LIN {X 0,Y 176.107,Z 395.866,A -85,B 0,C 180,E1 -22410,E2 -22410} C_VEL
LIN {X 0,Y 175.971,Z 396.64,A -85,B 0,C 180,E1 -22413.176,E2 -22413.176} C_VEL
LIN {X 0,Y 176.141,Z 396.55,A -85,B 0,C 180,E1 -22416.875,E2 -22416.875} C_VEL
LIN {X 0,Y 177.062,Z 394.985,A -85,B 0,C 180,E1 -22421.447,E2 -22421.447} C_VEL
LIN {X 0,Y 178.888,Z 391.863,A -85,B 0,C 180,E1 -22425.963,E2 -22425.963} C_VEL
LIN {X 0,Y 181.119,Z 388.376,A -85,B 0,C 180,E1 -22429.259,E2 -22429.259} C_VEL
LIN {X 0,Y 183.873,Z 383.839,A -85,B 0,C 180,E1 -22432.472,E2 -22432.472} C_VEL
LIN {X 0,Y 187.27,Z 377.805,A -85,B 0,C 180,E1 -22435.751,E2 -22435.751} C_VEL
LIN {X 0,Y 190.913,Z 371.032,A -85,B 0,C 180,E1 -22438.592,E2 -22438.592} C_VEL
LIN {X 0,Y 194.584,Z 363.85,A -85,B 0,C 180,E1 -22440.977,E2 -22440.977} C_VEL
LIN {X 0,Y 198.657,Z 355.185,A -85,B 0,C 180,E1 -22443.254,E2 -22443.254} C_VEL
LIN {X 0,Y 202.512,Z 345.804,A -85,B 0,C 180,E1 -22445.237,E2 -22445.237} C_VEL
LIN {X 0,Y 206.696,Z 334.241,A -85,B 0,C 180,E1 -22447.123,E2 -22447.123} C_VEL
LIN {X 0,Y 210.122,Z 322.779,A -85,B 0,C 180,E1 -22448.533,E2 -22448.533} C_VEL
LIN {X 0,Y 213.195,Z 309.844,A -85,B 0,C 180,E1 -22449.695,E2 -22449.695} C_VEL
LIN {X 0,Y 215.445,Z 296.998,A -85,B 0,C 180,E1 -22450.494,E2 -22450.494} C_VEL
LIN {X 0,Y 216.943,Z 281.701,A -85,B 0,C 180,E1 -22451.095,E2 -22451.095} C_VEL
LIN {X 0,Y 219.43,Z 248.273,A -85,B 0,C 180,E1 -22452.213,E2 -22452.213} C_VEL
LIN {X 0,Y 215.61,Z 238.212,A -85,B 0,C 180,E1 -22454.099,E2 -22454.099} C_VEL
LIN {X 0,Y 211.293,Z 228.849,A -85,B 0,C 180,E1 -22456.335,E2 -22456.335} C_VEL
LIN {X 0,Y 207.297,Z 221.367,A -85,B 0,C 180,E1 -22458.577,E2 -22458.577} C_VEL
LIN {X 0,Y 204.226,Z 216.042,A -85,B 0,C 180,E1 -22460.464,E2 -22460.464} C_VEL
LIN {X 0,Y 201.816,Z 212.042,A -85,B 0,C 180,E1 -22462.084,E2 -22462.084} C_VEL
LIN {X 0,Y 198.513,Z 206.797,A -85,B 0,C 180,E1 -22464.567,E2 -22464.567} C_VEL
LIN {X 0,Y 195.162,Z 201.691,A -85,B 0,C 180,E1 -22467.535,E2 -22467.535} C_VEL
LIN {X 0,Y 190.243,Z 194.896,A -85,B 0,C 180,E1 -22473.389,E2 -22473.389} C_VEL
LIN {X 0,Y 188.466,Z 192.868,A -85,B 0,C 180,E1 -22476.516,E2 -22476.516} C_VEL
LIN {X 0,Y 186.707,Z 191.554,A -85,B 0,C 180,E1 -22482.474,E2 -22482.474} C_VEL
LIN {X 0,Y 187.001,Z 191.732,A -85,B 0,C 180,E1 -22487.731,E2 -22487.731} C_VEL
LIN {X 0,Y 190.09,Z 193.411,A -85,B 0,C 180,E1 -22494.59,E2 -22494.59} C_VEL
LIN {X 0,Y 191.562,Z 196.122,A -85,B 0,C 180,E1 -22496.845,E2 -22496.845} C_VEL
LIN {X 0,Y 194.554,Z 198.965,A -85,B 0,C 180,E1 -22500.1,E2 -22500.1} C_VEL
LIN {X 0,Y 196.432,Z 202.226,A -85,B 0,C 180,E1 -22501.969,E2 -22501.969} C_VEL
LIN {X 0,Y 198.646,Z 204.552,A -85,B 0,C 180,E1 -22503.76,E2 -22503.76} C_VEL
LIN {X 0,Y 201.367,Z 208.221,A -85,B 0,C 180,E1 -22505.775,E2 -22505.775} C_VEL
LIN {X 0,Y 205.369,Z 214.172,A -85,B 0,C 180,E1 -22508.417,E2 -22508.417} C_VEL
LIN {X 0,Y 208.768,Z 219.318,A -85,B 0,C 180,E1 -22510.395,E2 -22510.395} C_VEL
LIN {X 0,Y 213.795,Z 228.478,A -85,B 0,C 180,E1 -22513.074,E2 -22513.074} C_VEL
LIN {X 0,Y 218.198,Z 237.802,A -85,B 0,C 180,E1 -22515.242,E2 -22515.242} C_VEL
LIN {X 0,Y 219.838,Z 242.158,A -85,B 0,C 180,E1 -22516.031,E2 -22516.031} C_VEL
LIN {X 0,Y 216.381,Z 285.399,A -85,B 0,C 180,E1 -22517.487,E2 -22517.487} C_VEL
LIN {X 0,Y 214.339,Z 299.301,A -85,B 0,C 180,E1 -22518.288,E2 -22518.288} C_VEL
LIN {X 0,Y 212.077,Z 310.584,A -85,B 0,C 180,E1 -22519.264,E2 -22519.264} C_VEL
LIN {X 0,Y 209.226,Z 321.582,A -85,B 0,C 180,E1 -22520.521,E2 -22520.521} C_VEL
LIN {X 0,Y 205.857,Z 332.053,A -85,B 0,C 180,E1 -22522.058,E2 -22522.058} C_VEL
LIN {X 0,Y 201.926,Z 342.352,A -85,B 0,C 180,E1 -22523.987,E2 -22523.987} C_VEL
LIN {X 0,Y 197.854,Z 351.744,A -85,B 0,C 180,E1 -22526.244,E2 -22526.244} C_VEL
LIN {X 0,Y 194.184,Z 359.384,A -85,B 0,C 180,E1 -22528.562,E2 -22528.562} C_VEL
LIN {X 0,Y 189.903,Z 367.38,A -85,B 0,C 180,E1 -22531.657,E2 -22531.657} C_VEL
LIN {X 0,Y 186.09,Z 373.869,A -85,B 0,C 180,E1 -22534.974,E2 -22534.974} C_VEL
LIN {X 0,Y 182.698,Z 379.213,A -85,B 0,C 180,E1 -22538.636,E2 -22538.636} C_VEL
LIN {X 0,Y 180.161,Z 382.905,A -85,B 0,C 180,E1 -22542.167,E2 -22542.167} C_VEL
LIN {X 0,Y 178.583,Z 385.029,A -85,B 0,C 180,E1 -22545.103,E2 -22545.103} C_VEL
LIN {X 0,Y 176.984,Z 386.777,A -85,B 0,C 180,E1 -22548.981,E2 -22548.981} C_VEL
LIN {X 0,Y 175.948,Z 387.352,A -85,B 0,C 180,E1 -22553.19,E2 -22553.19} C_VEL
LIN {X 0,Y 175.55,Z 386.619,A -85,B 0,C 180,E1 -22557.217,E2 -22557.217} C_VEL
LIN {X 0,Y 175.745,Z 384.409,A -85,B 0,C 180,E1 -22561.616,E2 -22561.616} C_VEL
LIN {X 0,Y 176.396,Z 381.454,A -85,B 0,C 180,E1 -22565.194,E2 -22565.194} C_VEL
LIN {X 0,Y 177.371,Z 376.912,A -85,B 0,C 180,E1 -22569.108,E2 -22569.108} C_VEL
LIN {X 0,Y 178.752,Z 371.021,A -85,B 0,C 180,E1 -22572.85,E2 -22572.85} C_VEL
LIN {X 0,Y 180.733,Z 363.522,A -85,B 0,C 180,E1 -22576.507,E2 -22576.507} C_VEL
LIN {X 0,Y 182.897,Z 355.757,A -85,B 0,C 180,E1 -22579.483,E2 -22579.483} C_VEL
LIN {X 0,Y 185.395,Z 346.038,A -85,B 0,C 180,E1 -22582.428,E2 -22582.428} C_VEL
LIN {X 0,Y 187.967,Z 335.639,A -85,B 0,C 180,E1 -22584.905,E2 -22584.905} C_VEL
LIN {X 0,Y 190.293,Z 324.879,A -85,B 0,C 180,E1 -22586.929,E2 -22586.929} C_VEL
LIN {X 0,Y 192.529,Z 312.621,A -85,B 0,C 180,E1 -22588.693,E2 -22588.693} C_VEL
LIN {X 0,Y 194.287,Z 300.473,A -85,B 0,C 180,E1 -22590,E2 -22590} C_VEL
LIN {X 0,Y 195.769,Z 287.395,A -85,B 0,C 180,E1 -22590.965,E2 -22590.965} C_VEL
LIN {X 0,Y 196.873,Z 270.105,A -85,B 0,C 180,E1 -22591.715,E2 -22591.715} C_VEL
LIN {X 0,Y 199.108,Z 225.699,A -85,B 0,C 180,E1 -22593.359,E2 -22593.359} C_VEL
LIN {X 0,Y 191.463,Z 205.022,A -85,B 0,C 180,E1 -22595.583,E2 -22595.583} C_VEL
LIN {X 0,Y 180.314,Z 184.581,A -85,B 0,C 180,E1 -22598.719,E2 -22598.719} C_VEL
LIN {X 0,Y 179.05,Z 182.009,A -85,B 0,C 180,E1 -22599.118,E2 -22599.118} C_VEL
LIN {X 0,Y 178.891,Z 181.212,A -85,B 0,C 180,E1 -22599.193,E2 -22599.193} C_VEL
LIN {X 0,Y 178.638,Z 181.233,A -85,B 0,C 180,E1 -22603.654,E2 -22603.654} C_VEL
LIN {X 0,Y 178.565,Z 181.241,A -85,B 0,C 180,E1 -22609.161,E2 -22609.161} C_VEL
LIN {X 0,Y 178.466,Z 181.238,A -85,B 0,C 180,E1 -22615.076,E2 -22615.076} C_VEL
LIN {X 0,Y 178.462,Z 181.246,A -85,B 0,C 180,E1 -22620.794,E2 -22620.794} C_VEL
LIN {X 0,Y 178.484,Z 181.225,A -85,B 0,C 180,E1 -22624.218,E2 -22624.218} C_VEL
LIN {X 0,Y 178.39,Z 181.264,A -85,B 0,C 180,E1 -22629.076,E2 -22629.076} C_VEL
LIN {X 0,Y 178.395,Z 181.255,A -85,B 0,C 180,E1 -22632.046,E2 -22632.046} C_VEL
LIN {X 0,Y 178.392,Z 181.224,A -85,B 0,C 180,E1 -22635.165,E2 -22635.165} C_VEL
LIN {X 0,Y 178.398,Z 181.233,A -85,B 0,C 180,E1 -22638.462,E2 -22638.462} C_VEL
LIN {X 0,Y 178.42,Z 181.26,A -85,B 0,C 180,E1 -22643.782,E2 -22643.782} C_VEL
LIN {X 0,Y 178.485,Z 181.245,A -85,B 0,C 180,E1 -22646.546,E2 -22646.546} C_VEL
LIN {X 0,Y 178.446,Z 181.256,A -85,B 0,C 180,E1 -22651.796,E2 -22651.796} C_VEL
LIN {X 0,Y 178.517,Z 181.241,A -85,B 0,C 180,E1 -22654.889,E2 -22654.889} C_VEL
LIN {X 0,Y 178.608,Z 181.235,A -85,B 0,C 180,E1 -22661.652,E2 -22661.652} C_VEL
LIN {X 0,Y 178.63,Z 181.221,A -85,B 0,C 180,E1 -22666.346,E2 -22666.346} C_VEL
LIN {X 0,Y 178.908,Z 181.197,A -85,B 0,C 180,E1 -22670.959,E2 -22670.959} C_VEL
LIN {X 0,Y 179.127,Z 181.171,A -85,B 0,C 180,E1 -22677.751,E2 -22677.751} C_VEL
LIN {X 0,Y 179.347,Z 181.143,A -85,B 0,C 180,E1 -22680,E2 -22680} C_VEL
LIN {X 0,Y 178.834,Z 181.175,A -85,B 0,C 180,E1 -22684.508,E2 -22684.508} C_VEL
LIN {X 0,Y 178.905,Z 181.171,A -85,B 0,C 180,E1 -22689.04,E2 -22689.04} C_VEL
LIN {X 0,Y 178.625,Z 181.235,A -85,B 0,C 180,E1 -22693.655,E2 -22693.655} C_VEL
LIN {X 0,Y 178.555,Z 181.214,A -85,B 0,C 180,E1 -22699.151,E2 -22699.151} C_VEL
LIN {X 0,Y 178.506,Z 181.248,A -85,B 0,C 180,E1 -22705.103,E2 -22705.103} C_VEL
LIN {X 0,Y 178.461,Z 181.256,A -85,B 0,C 180,E1 -22710.794,E2 -22710.794} C_VEL
LIN {X 0,Y 178.484,Z 181.249,A -85,B 0,C 180,E1 -22714.218,E2 -22714.218} C_VEL
LIN {X 0,Y 178.388,Z 181.265,A -85,B 0,C 180,E1 -22719.076,E2 -22719.076} C_VEL
LIN {X 0,Y 178.394,Z 181.262,A -85,B 0,C 180,E1 -22722.046,E2 -22722.046} C_VEL
LIN {X 0,Y 178.431,Z 181.452,A -85,B 0,C 180,E1 -22726.724,E2 -22726.724} C_VEL
LIN {X 0,Y 179.299,Z 184.858,A -85,B 0,C 180,E1 -22728.666,E2 -22728.666} C_VEL
LIN {X 0,Y 186.421,Z 200.095,A -85,B 0,C 180,E1 -22730.858,E2 -22730.858} C_VEL
LIN {X 0,Y 193.884,Z 218.787,A -85,B 0,C 180,E1 -22733.074,E2 -22733.074} C_VEL
LIN {X 0,Y 196.789,Z 227.908,A -85,B 0,C 180,E1 -22733.967,E2 -22733.967} C_VEL
LIN {X 0,Y 198.481,Z 242.952,A -85,B 0,C 180,E1 -22734.906,E2 -22734.906} C_VEL
LIN {X 0,Y 195.784,Z 293.869,A -85,B 0,C 180,E1 -22736.844,E2 -22736.844} C_VEL
LIN {X 0,Y 194.316,Z 307.658,A -85,B 0,C 180,E1 -22737.759,E2 -22737.759} C_VEL
LIN {X 0,Y 193.602,Z 312.687,A -85,B 0,C 180,E1 -22738.205,E2 -22738.205} C_VEL
LIN {X 0,Y 192.145,Z 318.194,A -85,B 0,C 180,E1 -22738.68,E2 -22738.68} C_VEL
LIN {X 0,Y 188.016,Z 326.878,A -85,B 0,C 180,E1 -22739.416,E2 -22739.416} C_VEL
LIN {X 0,Y 183.577,Z 335.199,A -85,B 0,C 180,E1 -22740.384,E2 -22740.384} C_VEL
LIN {X 0,Y 181.663,Z 340.142,A -85,B 0,C 180,E1 -22741.217,E2 -22741.217} C_VEL
LIN {X 0,Y 179.121,Z 350.496,A -85,B 0,C 180,E1 -22743.493,E2 -22743.493} C_VEL
LIN {X 0,Y 176.758,Z 359.609,A -85,B 0,C 180,E1 -22746.012,E2 -22746.012} C_VEL
LIN {X 0,Y 175.261,Z 365.095,A -85,B 0,C 180,E1 -22747.815,E2 -22747.815} C_VEL
LIN {X 0,Y 173.041,Z 373.154,A -85,B 0,C 180,E1 -22751.039,E2 -22751.039} C_VEL
LIN {X 0,Y 171.159,Z 380.029,A -85,B 0,C 180,E1 -22754.52,E2 -22754.52} C_VEL
LIN {X 0,Y 169.97,Z 385.517,A -85,B 0,C 180,E1 -22758.068,E2 -22758.068} C_VEL
LIN {X 0,Y 169.249,Z 389.772,A -85,B 0,C 180,E1 -22761.643,E2 -22761.643} C_VEL
LIN {X 0,Y 168.931,Z 392.919,A -85,B 0,C 180,E1 -22765.227,E2 -22765.227} C_VEL
LIN {X 0,Y 168.947,Z 394.472,A -85,B 0,C 180,E1 -22767.616,E2 -22767.616} C_VEL
LIN {X 0,Y 169.015,Z 395.567,A -85,B 0,C 180,E1 -22770,E2 -22770} C_VEL
LIN {X 0,Y 168.892,Z 396.323,A -85,B 0,C 180,E1 -22772.921,E2 -22772.921} C_VEL
LIN {X 0,Y 169.093,Z 396.381,A -85,B 0,C 180,E1 -22777.163,E2 -22777.163} C_VEL
LIN {X 0,Y 169.462,Z 395.868,A -85,B 0,C 180,E1 -22779.549,E2 -22779.549} C_VEL
LIN {X 0,Y 170.961,Z 393.626,A -85,B 0,C 180,E1 -22784.28,E2 -22784.28} C_VEL
LIN {X 0,Y 172.77,Z 390.889,A -85,B 0,C 180,E1 -22787.764,E2 -22787.764} C_VEL
LIN {X 0,Y 175.373,Z 387.162,A -85,B 0,C 180,E1 -22791.142,E2 -22791.142} C_VEL
LIN {X 0,Y 178.401,Z 382.356,A -85,B 0,C 180,E1 -22794.434,E2 -22794.434} C_VEL
LIN {X 0,Y 182.612,Z 375.225,A -85,B 0,C 180,E1 -22798.129,E2 -22798.129} C_VEL
LIN {X 0,Y 186.944,Z 367.53,A -85,B 0,C 180,E1 -22801.126,E2 -22801.126} C_VEL
LIN {X 0,Y 191.916,Z 357.942,A -85,B 0,C 180,E1 -22803.95,E2 -22803.95} C_VEL
LIN {X 0,Y 196.347,Z 348.123,A -85,B 0,C 180,E1 -22806.2,E2 -22806.2} C_VEL
LIN {X 0,Y 200.691,Z 337.124,A -85,B 0,C 180,E1 -22808.113,E2 -22808.113} C_VEL
LIN {X 0,Y 204.719,Z 324.761,A -85,B 0,C 180,E1 -22809.747,E2 -22809.747} C_VEL
LIN {X 0,Y 207.863,Z 312.663,A -85,B 0,C 180,E1 -22810.926,E2 -22810.926} C_VEL
LIN {X 0,Y 210.488,Z 299.25,A -85,B 0,C 180,E1 -22811.816,E2 -22811.816} C_VEL
LIN {X 0,Y 212.045,Z 286.37,A -85,B 0,C 180,E1 -22812.391,E2 -22812.391} C_VEL
LIN {X 0,Y 214.842,Z 250.537,A -85,B 0,C 180,E1 -22813.61,E2 -22813.61} C_VEL
LIN {X 0,Y 211.062,Z 240.778,A -85,B 0,C 180,E1 -22815.632,E2 -22815.632} C_VEL
LIN {X 0,Y 206.868,Z 231.538,A -85,B 0,C 180,E1 -22818.017,E2 -22818.017} C_VEL
LIN {X 0,Y 202.25,Z 222.91,A -85,B 0,C 180,E1 -22820.911,E2 -22820.911} C_VEL
LIN {X 0,Y 199.146,Z 217.613,A -85,B 0,C 180,E1 -22823.134,E2 -22823.134} C_VEL
LIN {X 0,Y 196.249,Z 212.847,A -85,B 0,C 180,E1 -22825.454,E2 -22825.454} C_VEL
LIN {X 0,Y 192.831,Z 207.539,A -85,B 0,C 180,E1 -22828.749,E2 -22828.749} C_VEL
LIN {X 0,Y 188.741,Z 201.564,A -85,B 0,C 180,E1 -22834.1,E2 -22834.1} C_VEL
LIN {X 0,Y 187.288,Z 199.823,A -85,B 0,C 180,E1 -22836.895,E2 -22836.895} C_VEL
LIN {X 0,Y 185.731,Z 198.59,A -85,B 0,C 180,E1 -22842.379,E2 -22842.379} C_VEL
LIN {X 0,Y 186.009,Z 198.77,A -85,B 0,C 180,E1 -22847.752,E2 -22847.752} C_VEL
LIN {X 0,Y 188.742,Z 200.32,A -85,B 0,C 180,E1 -22854.119,E2 -22854.119} C_VEL
LIN {X 0,Y 190.143,Z 202.883,A -85,B 0,C 180,E1 -22856.351,E2 -22856.351} C_VEL
LIN {X 0,Y 192.838,Z 205.635,A -85,B 0,C 180,E1 -22859.478,E2 -22859.478} C_VEL
LIN {X 0,Y 194.729,Z 208.869,A -85,B 0,C 180,E1 -22861.431,E2 -22861.431} C_VEL
LIN {X 0,Y 196.672,Z 211.096,A -85,B 0,C 180,E1 -22863.118,E2 -22863.118} C_VEL
LIN {X 0,Y 199.963,Z 215.717,A -85,B 0,C 180,E1 -22865.637,E2 -22865.637} C_VEL
LIN {X 0,Y 204.862,Z 223.149,A -85,B 0,C 180,E1 -22868.874,E2 -22868.874} C_VEL
LIN {X 0,Y 208.76,Z 230.33,A -85,B 0,C 180,E1 -22871.187,E2 -22871.187} C_VEL
LIN {X 0,Y 212.936,Z 238.93,A -85,B 0,C 180,E1 -22873.425,E2 -22873.425} C_VEL
LIN {X 0,Y 215.288,Z 244.559,A -85,B 0,C 180,E1 -22874.639,E2 -22874.639} C_VEL
LIN {X 0,Y 211.784,Z 285.821,A -85,B 0,C 180,E1 -22876.042,E2 -22876.042} C_VEL
LIN {X 0,Y 209.706,Z 299.278,A -85,B 0,C 180,E1 -22876.818,E2 -22876.818} C_VEL
LIN {X 0,Y 207.25,Z 311.125,A -85,B 0,C 180,E1 -22877.853,E2 -22877.853} C_VEL
LIN {X 0,Y 203.846,Z 323.371,A -85,B 0,C 180,E1 -22879.297,E2 -22879.297} C_VEL
LIN {X 0,Y 199.706,Z 335.316,A -85,B 0,C 180,E1 -22881.158,E2 -22881.158} C_VEL
LIN {X 0,Y 195.305,Z 345.853,A -85,B 0,C 180,E1 -22883.318,E2 -22883.318} C_VEL
LIN {X 0,Y 191.287,Z 354.267,A -85,B 0,C 180,E1 -22885.521,E2 -22885.521} C_VEL
LIN {X 0,Y 187.201,Z 361.997,A -85,B 0,C 180,E1 -22888.084,E2 -22888.084} C_VEL
LIN {X 0,Y 182.843,Z 369.539,A -85,B 0,C 180,E1 -22891.316,E2 -22891.316} C_VEL
LIN {X 0,Y 179.147,Z 375.283,A -85,B 0,C 180,E1 -22894.528,E2 -22894.528} C_VEL
LIN {X 0,Y 175.416,Z 380.612,A -85,B 0,C 180,E1 -22898.623,E2 -22898.623} C_VEL
LIN {X 0,Y 172.573,Z 384.364,A -85,B 0,C 180,E1 -22902.857,E2 -22902.857} C_VEL
LIN {X 0,Y 171.125,Z 386.009,A -85,B 0,C 180,E1 -22905.718,E2 -22905.718} C_VEL
LIN {X 0,Y 170.001,Z 387.077,A -85,B 0,C 180,E1 -22908.589,E2 -22908.589} C_VEL
LIN {X 0,Y 169.019,Z 387.547,A -85,B 0,C 180,E1 -22912.19,E2 -22912.19} C_VEL
LIN {X 0,Y 168.488,Z 386.939,A -85,B 0,C 180,E1 -22916.537,E2 -22916.537} C_VEL
LIN {X 0,Y 168.576,Z 384.833,A -85,B 0,C 180,E1 -22921.105,E2 -22921.105} C_VEL
LIN {X 0,Y 169.348,Z 381.387,A -85,B 0,C 180,E1 -22925.48,E2 -22925.48} C_VEL
LIN {X 0,Y 170.352,Z 376.838,A -85,B 0,C 180,E1 -22929.471,E2 -22929.471} C_VEL
LIN {X 0,Y 171.814,Z 370.863,A -85,B 0,C 180,E1 -22933.361,E2 -22933.361} C_VEL
LIN {X 0,Y 173.965,Z 363.113,A -85,B 0,C 180,E1 -22937.235,E2 -22937.235} C_VEL
LIN {X 0,Y 176.178,Z 355.408,A -85,B 0,C 180,E1 -22940.239,E2 -22940.239} C_VEL
LIN {X 0,Y 178.778,Z 345.747,A -85,B 0,C 180,E1 -22943.227,E2 -22943.227} C_VEL
LIN {X 0,Y 181.436,Z 335.304,A -85,B 0,C 180,E1 -22945.772,E2 -22945.772} C_VEL
LIN {X 0,Y 183.793,Z 324.677,A -85,B 0,C 180,E1 -22947.808,E2 -22947.808} C_VEL
LIN {X 0,Y 186.077,Z 312.539,A -85,B 0,C 180,E1 -22949.594,E2 -22949.594} C_VEL
LIN {X 0,Y 187.926,Z 300.289,A -85,B 0,C 180,E1 -22950.937,E2 -22950.937} C_VEL
LIN {X 0,Y 189.456,Z 286.987,A -85,B 0,C 180,E1 -22951.927,E2 -22951.927} C_VEL
LIN {X 0,Y 190.6,Z 269.299,A -85,B 0,C 180,E1 -22952.701,E2 -22952.701} C_VEL
LIN {X 0,Y 192.875,Z 227.779,A -85,B 0,C 180,E1 -22954.266,E2 -22954.266} C_VEL
LIN {X 0,Y 185.991,Z 208.623,A -85,B 0,C 180,E1 -22956.403,E2 -22956.403} C_VEL
LIN {X 0,Y 174.96,Z 188.375,A -85,B 0,C 180,E1 -22959.659,E2 -22959.659} C_VEL
LIN {X 0,Y 173.38,Z 185.708,A -85,B 0,C 180,E1 -22960.157,E2 -22960.157} C_VEL
LIN {X 0,Y 172.041,Z 183.219,A -85,B 0,C 180,E1 -22960.601,E2 -22960.601} C_VEL
LIN {X 0,Y 171.798,Z 182.075,A -85,B 0,C 180,E1 -22960.758,E2 -22960.758} C_VEL
LIN {X 0,Y 171.517,Z 182.104,A -85,B 0,C 180,E1 -22966.668,E2 -22966.668} C_VEL
LIN {X 0,Y 171.491,Z 182.124,A -85,B 0,C 180,E1 -22969.51,E2 -22969.51} C_VEL
LIN {X 0,Y 171.404,Z 182.121,A -85,B 0,C 180,E1 -22975.57,E2 -22975.57} C_VEL
LIN {X 0,Y 171.419,Z 182.125,A -85,B 0,C 180,E1 -22980.573,E2 -22980.573} C_VEL
LIN {X 0,Y 171.393,Z 182.112,A -85,B 0,C 180,E1 -22985.035,E2 -22985.035} C_VEL
LIN {X 0,Y 171.353,Z 182.14,A -85,B 0,C 180,E1 -22988.805,E2 -22988.805} C_VEL
LIN {X 0,Y 171.319,Z 182.113,A -85,B 0,C 180,E1 -22994.218,E2 -22994.218} C_VEL
LIN {X 0,Y 171.331,Z 182.118,A -85,B 0,C 180,E1 -22998.98,E2 -22998.98} C_VEL
LIN {X 0,Y 171.361,Z 182.136,A -85,B 0,C 180,E1 -23002.034,E2 -23002.034} C_VEL
LIN {X 0,Y 171.399,Z 182.133,A -85,B 0,C 180,E1 -23005.093,E2 -23005.093} C_VEL
LIN {X 0,Y 171.411,Z 182.129,A -85,B 0,C 180,E1 -23010.527,E2 -23010.527} C_VEL
LIN {X 0,Y 171.438,Z 182.119,A -85,B 0,C 180,E1 -23015.798,E2 -23015.798} C_VEL
LIN {X 0,Y 171.509,Z 182.121,A -85,B 0,C 180,E1 -23020.863,E2 -23020.863} C_VEL
LIN {X 0,Y 171.545,Z 182.101,A -85,B 0,C 180,E1 -23025.77,E2 -23025.77} C_VEL
LIN {X 0,Y 171.846,Z 182.078,A -85,B 0,C 180,E1 -23030.585,E2 -23030.585} C_VEL
LIN {X 0,Y 171.787,Z 182.077,A -85,B 0,C 180,E1 -23035.307,E2 -23035.307} C_VEL
LIN {X 0,Y 172.312,Z 182.019,A -85,B 0,C 180,E1 -23040,E2 -23040} C_VEL
LIN {X 0,Y 171.783,Z 182.048,A -85,B 0,C 180,E1 -23044.693,E2 -23044.693} C_VEL
LIN {X 0,Y 171.844,Z 182.054,A -85,B 0,C 180,E1 -23049.415,E2 -23049.415} C_VEL
LIN {X 0,Y 171.541,Z 182.117,A -85,B 0,C 180,E1 -23054.23,E2 -23054.23} C_VEL
LIN {X 0,Y 171.479,Z 182.092,A -85,B 0,C 180,E1 -23059.498,E2 -23059.498} C_VEL
LIN {X 0,Y 171.436,Z 182.131,A -85,B 0,C 180,E1 -23065.592,E2 -23065.592} C_VEL
LIN {X 0,Y 171.419,Z 182.133,A -85,B 0,C 180,E1 -23070.572,E2 -23070.572} C_VEL
LIN {X 0,Y 171.393,Z 182.135,A -85,B 0,C 180,E1 -23075.035,E2 -23075.035} C_VEL
LIN {X 0,Y 171.344,Z 182.143,A -85,B 0,C 180,E1 -23078.801,E2 -23078.801} C_VEL
LIN {X 0,Y 171.319,Z 182.137,A -85,B 0,C 180,E1 -23084.218,E2 -23084.218} C_VEL
LIN {X 0,Y 171.386,Z 182.139,A -85,B 0,C 180,E1 -23085.599,E2 -23085.599} C_VEL
LIN {X 0,Y 171.959,Z 184.583,A -85,B 0,C 180,E1 -23087.052,E2 -23087.052} C_VEL
LIN {X 0,Y 178.775,Z 198.802,A -85,B 0,C 180,E1 -23089.287,E2 -23089.287} C_VEL
LIN {X 0,Y 185.122,Z 213.873,A -85,B 0,C 180,E1 -23091.293,E2 -23091.293} C_VEL
LIN {X 0,Y 190.538,Z 228.94,A -85,B 0,C 180,E1 -23092.988,E2 -23092.988} C_VEL
LIN {X 0,Y 192.183,Z 243.751,A -85,B 0,C 180,E1 -23093.956,E2 -23093.956} C_VEL
LIN {X 0,Y 189.431,Z 293.655,A -85,B 0,C 180,E1 -23095.91,E2 -23095.91} C_VEL
LIN {X 0,Y 187.93,Z 307.365,A -85,B 0,C 180,E1 -23096.843,E2 -23096.843} C_VEL
LIN {X 0,Y 186.046,Z 319.586,A -85,B 0,C 180,E1 -23098.071,E2 -23098.071} C_VEL
LIN {X 0,Y 183.534,Z 332.205,A -85,B 0,C 180,E1 -23099.828,E2 -23099.828} C_VEL
LIN {X 0,Y 181.663,Z 340.142,A -85,B 0,C 180,E1 -23101.217,E2 -23101.217} C_VEL
LIN {X 0,Y 179.676,Z 345.025,A -85,B 0,C 180,E1 -23102.13,E2 -23102.13} C_VEL
LIN {X 0,Y 172.868,Z 355.309,A -85,B 0,C 180,E1 -23104.252,E2 -23104.252} C_VEL
LIN {X 0,Y 169.601,Z 360.842,A -85,B 0,C 180,E1 -23105.784,E2 -23105.784} C_VEL
LIN {X 0,Y 168.69,Z 363.503,A -85,B 0,C 180,E1 -23106.693,E2 -23106.693} C_VEL
LIN {X 0,Y 167.072,Z 369.581,A -85,B 0,C 180,E1 -23109.05,E2 -23109.05} C_VEL
LIN {X 0,Y 164.926,Z 377.141,A -85,B 0,C 180,E1 -23112.645,E2 -23112.645} C_VEL
LIN {X 0,Y 163.342,Z 383.188,A -85,B 0,C 180,E1 -23116.311,E2 -23116.311} C_VEL
LIN {X 0,Y 162.414,Z 387.947,A -85,B 0,C 180,E1 -23120.033,E2 -23120.033} C_VEL
LIN {X 0,Y 161.906,Z 391.539,A -85,B 0,C 180,E1 -23123.77,E2 -23123.77} C_VEL
LIN {X 0,Y 161.866,Z 394.085,A -85,B 0,C 180,E1 -23127.512,E2 -23127.512} C_VEL
LIN {X 0,Y 161.924,Z 395.256,A -85,B 0,C 180,E1 -23130,E2 -23130} C_VEL
LIN {X 0,Y 161.797,Z 395.963,A -85,B 0,C 180,E1 -23132.49,E2 -23132.49} C_VEL
LIN {X 0,Y 161.85,Z 396.276,A -85,B 0,C 180,E1 -23134.982,E2 -23134.982} C_VEL
LIN {X 0,Y 162.44,Z 395.758,A -85,B 0,C 180,E1 -23139.966,E2 -23139.966} C_VEL
LIN {X 0,Y 163.131,Z 394.899,A -85,B 0,C 180,E1 -23142.44,E2 -23142.44} C_VEL
LIN {X 0,Y 165.232,Z 391.971,A -85,B 0,C 180,E1 -23147.322,E2 -23147.322} C_VEL
LIN {X 0,Y 167.763,Z 388.674,A -85,B 0,C 180,E1 -23150.86,E2 -23150.86} C_VEL
LIN {X 0,Y 170.809,Z 384.361,A -85,B 0,C 180,E1 -23154.296,E2 -23154.296} C_VEL
LIN {X 0,Y 174.933,Z 378.091,A -85,B 0,C 180,E1 -23158.048,E2 -23158.048} C_VEL
LIN {X 0,Y 179.394,Z 370.883,A -85,B 0,C 180,E1 -23161.271,E2 -23161.271} C_VEL
LIN {X 0,Y 183.502,Z 363.774,A -85,B 0,C 180,E1 -23163.735,E2 -23163.735} C_VEL
LIN {X 0,Y 187.957,Z 355.211,A -85,B 0,C 180,E1 -23166.08,E2 -23166.08} C_VEL
LIN {X 0,Y 192.215,Z 345.901,A -85,B 0,C 180,E1 -23168.098,E2 -23168.098} C_VEL
LIN {X 0,Y 196.761,Z 334.474,A -85,B 0,C 180,E1 -23170.011,E2 -23170.011} C_VEL
LIN {X 0,Y 200.465,Z 323.297,A -85,B 0,C 180,E1 -23171.432,E2 -23171.432} C_VEL
LIN {X 0,Y 203.774,Z 310.711,A -85,B 0,C 180,E1 -23172.598,E2 -23172.598} C_VEL
LIN {X 0,Y 206.365,Z 297.392,A -85,B 0,C 180,E1 -23173.453,E2 -23173.453} C_VEL
LIN {X 0,Y 207.997,Z 282.871,A -85,B 0,C 180,E1 -23174.052,E2 -23174.052} C_VEL
LIN {X 0,Y 210.445,Z 253.266,A -85,B 0,C 180,E1 -23175.05,E2 -23175.05} C_VEL
LIN {X 0,Y 207.149,Z 244.462,A -85,B 0,C 180,E1 -23176.956,E2 -23176.956} C_VEL
LIN {X 0,Y 203.33,Z 235.89,A -85,B 0,C 180,E1 -23179.332,E2 -23179.332} C_VEL
LIN {X 0,Y 199.096,Z 227.688,A -85,B 0,C 180,E1 -23182.237,E2 -23182.237} C_VEL
LIN {X 0,Y 196.6,Z 223.285,A -85,B 0,C 180,E1 -23184.167,E2 -23184.167} C_VEL
LIN {X 0,Y 194.365,Z 219.331,A -85,B 0,C 180,E1 -23186.106,E2 -23186.106} C_VEL
LIN {X 0,Y 191.155,Z 214.149,A -85,B 0,C 180,E1 -23189.363,E2 -23189.363} C_VEL
LIN {X 0,Y 187.361,Z 208.322,A -85,B 0,C 180,E1 -23194.669,E2 -23194.669} C_VEL
LIN {X 0,Y 186.118,Z 206.776,A -85,B 0,C 180,E1 -23197.279,E2 -23197.279} C_VEL
LIN {X 0,Y 184.756,Z 205.624,A -85,B 0,C 180,E1 -23202.283,E2 -23202.283} C_VEL
LIN {X 0,Y 185.007,Z 205.776,A -85,B 0,C 180,E1 -23207.685,E2 -23207.685} C_VEL
LIN {X 0,Y 187.517,Z 207.361,A -85,B 0,C 180,E1 -23213.812,E2 -23213.812} C_VEL
LIN {X 0,Y 189.221,Z 210.259,A -85,B 0,C 180,E1 -23216.523,E2 -23216.523} C_VEL
LIN {X 0,Y 191.172,Z 212.351,A -85,B 0,C 180,E1 -23218.881,E2 -23218.881} C_VEL
LIN {X 0,Y 193.376,Z 215.915,A -85,B 0,C 180,E1 -23221.2,E2 -23221.2} C_VEL
LIN {X 0,Y 194.887,Z 217.786,A -85,B 0,C 180,E1 -23222.565,E2 -23222.565} C_VEL
LIN {X 0,Y 197.754,Z 221.997,A -85,B 0,C 180,E1 -23224.895,E2 -23224.895} C_VEL
LIN {X 0,Y 202.144,Z 228.943,A -85,B 0,C 180,E1 -23227.994,E2 -23227.994} C_VEL
LIN {X 0,Y 205.659,Z 235.617,A -85,B 0,C 180,E1 -23230.199,E2 -23230.199} C_VEL
LIN {X 0,Y 209.687,Z 244.391,A -85,B 0,C 180,E1 -23232.533,E2 -23232.533} C_VEL
LIN {X 0,Y 210.887,Z 247.219,A -85,B 0,C 180,E1 -23233.186,E2 -23233.186} C_VEL
LIN {X 0,Y 207.416,Z 286.223,A -85,B 0,C 180,E1 -23234.52,E2 -23234.52} C_VEL
LIN {X 0,Y 205.186,Z 299.973,A -85,B 0,C 180,E1 -23235.319,E2 -23235.319} C_VEL
LIN {X 0,Y 202.714,Z 311.154,A -85,B 0,C 180,E1 -23236.299,E2 -23236.299} C_VEL
LIN {X 0,Y 199.234,Z 323.283,A -85,B 0,C 180,E1 -23237.742,E2 -23237.742} C_VEL
LIN {X 0,Y 195.19,Z 334.464,A -85,B 0,C 180,E1 -23239.471,E2 -23239.471} C_VEL
LIN {X 0,Y 190.532,Z 345.267,A -85,B 0,C 180,E1 -23241.646,E2 -23241.646} C_VEL
LIN {X 0,Y 186.342,Z 353.743,A -85,B 0,C 180,E1 -23243.849,E2 -23243.849} C_VEL
LIN {X 0,Y 181.27,Z 362.828,A -85,B 0,C 180,E1 -23246.907,E2 -23246.907} C_VEL
LIN {X 0,Y 176.91,Z 369.861,A -85,B 0,C 180,E1 -23250.013,E2 -23250.013} C_VEL
LIN {X 0,Y 172.79,Z 375.846,A -85,B 0,C 180,E1 -23253.507,E2 -23253.507} C_VEL
LIN {X 0,Y 168.831,Z 381.067,A -85,B 0,C 180,E1 -23257.727,E2 -23257.727} C_VEL
LIN {X 0,Y 166.726,Z 383.673,A -85,B 0,C 180,E1 -23260.645,E2 -23260.645} C_VEL
LIN {X 0,Y 164.978,Z 385.602,A -85,B 0,C 180,E1 -23263.598,E2 -23263.598} C_VEL
LIN {X 0,Y 163.414,Z 387.024,A -85,B 0,C 180,E1 -23266.981,E2 -23266.981} C_VEL
LIN {X 0,Y 162.113,Z 387.737,A -85,B 0,C 180,E1 -23271.293,E2 -23271.293} C_VEL
LIN {X 0,Y 161.422,Z 387.22,A -85,B 0,C 180,E1 -23275.815,E2 -23275.815} C_VEL
LIN {X 0,Y 161.423,Z 385.243,A -85,B 0,C 180,E1 -23280.547,E2 -23280.547} C_VEL
LIN {X 0,Y 162.004,Z 382.624,A -85,B 0,C 180,E1 -23284.29,E2 -23284.29} C_VEL
LIN {X 0,Y 162.951,Z 378.413,A -85,B 0,C 180,E1 -23288.494,E2 -23288.494} C_VEL
LIN {X 0,Y 164.302,Z 372.882,A -85,B 0,C 180,E1 -23292.577,E2 -23292.577} C_VEL
LIN {X 0,Y 166.239,Z 365.914,A -85,B 0,C 180,E1 -23296.499,E2 -23296.499} C_VEL
LIN {X 0,Y 168.537,Z 358.387,A -85,B 0,C 180,E1 -23299.792,E2 -23299.792} C_VEL
LIN {X 0,Y 171.059,Z 349.428,A -85,B 0,C 180,E1 -23302.92,E2 -23302.92} C_VEL
LIN {X 0,Y 173.774,Z 339.523,A -85,B 0,C 180,E1 -23305.651,E2 -23305.651} C_VEL
LIN {X 0,Y 176.456,Z 328.563,A -85,B 0,C 180,E1 -23308.003,E2 -23308.003} C_VEL
LIN {X 0,Y 178.953,Z 316.549,A -85,B 0,C 180,E1 -23310,E2 -23310} C_VEL
LIN {X 0,Y 181.042,Z 304.212,A -85,B 0,C 180,E1 -23311.529,E2 -23311.529} C_VEL
LIN {X 0,Y 182.811,Z 290.472,A -85,B 0,C 180,E1 -23312.708,E2 -23312.708} C_VEL
LIN {X 0,Y 183.913,Z 277.095,A -85,B 0,C 180,E1 -23313.418,E2 -23313.418} C_VEL
LIN {X 0,Y 186.533,Z 229.01,A -85,B 0,C 180,E1 -23315.304,E2 -23315.304} C_VEL
LIN {X 0,Y 180.356,Z 211.924,A -85,B 0,C 180,E1 -23317.301,E2 -23317.301} C_VEL
LIN {X 0,Y 169.034,Z 190.907,A -85,B 0,C 180,E1 -23320.865,E2 -23320.865} C_VEL
LIN {X 0,Y 166.42,Z 186.855,A -85,B 0,C 180,E1 -23321.715,E2 -23321.715} C_VEL
LIN {X 0,Y 164.829,Z 184.145,A -85,B 0,C 180,E1 -23322.264,E2 -23322.264} C_VEL
LIN {X 0,Y 164.589,Z 182.976,A -85,B 0,C 180,E1 -23322.484,E2 -23322.484} C_VEL
LIN {X 0,Y 164.44,Z 182.987,A -85,B 0,C 180,E1 -23327.408,E2 -23327.408} C_VEL
LIN {X 0,Y 164.423,Z 183.007,A -85,B 0,C 180,E1 -23329.996,E2 -23329.996} C_VEL
LIN {X 0,Y 164.34,Z 183.003,A -85,B 0,C 180,E1 -23336.094,E2 -23336.094} C_VEL
LIN {X 0,Y 164.354,Z 182.997,A -85,B 0,C 180,E1 -23341.215,E2 -23341.215} C_VEL
LIN {X 0,Y 164.293,Z 183.012,A -85,B 0,C 180,E1 -23346.79,E2 -23346.79} C_VEL
LIN {X 0,Y 164.289,Z 183.02,A -85,B 0,C 180,E1 -23349.917,E2 -23349.917} C_VEL
LIN {X 0,Y 164.281,Z 183,A -85,B 0,C 180,E1 -23353.342,E2 -23353.342} C_VEL
LIN {X 0,Y 164.261,Z 182.976,A -85,B 0,C 180,E1 -23356.798,E2 -23356.798} C_VEL
LIN {X 0,Y 164.29,Z 183.006,A -85,B 0,C 180,E1 -23360.355,E2 -23360.355} C_VEL
LIN {X 0,Y 164.327,Z 183.015,A -85,B 0,C 180,E1 -23364.351,E2 -23364.351} C_VEL
LIN {X 0,Y 164.369,Z 182.999,A -85,B 0,C 180,E1 -23369.13,E2 -23369.13} C_VEL
LIN {X 0,Y 164.396,Z 183,A -85,B 0,C 180,E1 -23374.69,E2 -23374.69} C_VEL
LIN {X 0,Y 164.418,Z 183.002,A -85,B 0,C 180,E1 -23380.117,E2 -23380.117} C_VEL
LIN {X 0,Y 164.475,Z 182.981,A -85,B 0,C 180,E1 -23385.144,E2 -23385.144} C_VEL
LIN {X 0,Y 164.767,Z 182.961,A -85,B 0,C 180,E1 -23390.176,E2 -23390.176} C_VEL
LIN {X 0,Y 164.824,Z 182.944,A -85,B 0,C 180,E1 -23392.651,E2 -23392.651} C_VEL
LIN {X 0,Y 165.276,Z 182.895,A -85,B 0,C 180,E1 -23400,E2 -23400} C_VEL
LIN {X 0,Y 164.821,Z 182.905,A -85,B 0,C 180,E1 -23407.349,E2 -23407.349} C_VEL
LIN {X 0,Y 164.703,Z 182.958,A -85,B 0,C 180,E1 -23411.057,E2 -23411.057} C_VEL
LIN {X 0,Y 164.429,Z 182.987,A -85,B 0,C 180,E1 -23417.409,E2 -23417.409} C_VEL
LIN {X 0,Y 164.421,Z 182.968,A -85,B 0,C 180,E1 -23419.996,E2 -23419.996} C_VEL
LIN {X 0,Y 164.365,Z 183.011,A -85,B 0,C 180,E1 -23426.112,E2 -23426.112} C_VEL
LIN {X 0,Y 164.358,Z 183.014,A -85,B 0,C 180,E1 -23431.217,E2 -23431.217} C_VEL
LIN {X 0,Y 164.281,Z 183.024,A -85,B 0,C 180,E1 -23436.793,E2 -23436.793} C_VEL
LIN {X 0,Y 164.286,Z 183.021,A -85,B 0,C 180,E1 -23439.918,E2 -23439.918} C_VEL
LIN {X 0,Y 164.321,Z 183.131,A -85,B 0,C 180,E1 -23444.562,E2 -23444.562} C_VEL
LIN {X 0,Y 164.662,Z 184.492,A -85,B 0,C 180,E1 -23445.308,E2 -23445.308} C_VEL
LIN {X 0,Y 172.92,Z 201.319,A -85,B 0,C 180,E1 -23448.184,E2 -23448.184} C_VEL
LIN {X 0,Y 179.484,Z 217.066,A -85,B 0,C 180,E1 -23450.379,E2 -23450.379} C_VEL
LIN {X 0,Y 184.558,Z 231.274,A -85,B 0,C 180,E1 -23452.045,E2 -23452.045} C_VEL
LIN {X 0,Y 185.96,Z 244.269,A -85,B 0,C 180,E1 -23452.934,E2 -23452.934} C_VEL
LIN {X 0,Y 183.106,Z 293.787,A -85,B 0,C 180,E1 -23454.933,E2 -23454.933} C_VEL
LIN {X 0,Y 181.483,Z 307.806,A -85,B 0,C 180,E1 -23455.923,E2 -23455.923} C_VEL
LIN {X 0,Y 179.638,Z 319.319,A -85,B 0,C 180,E1 -23457.123,E2 -23457.123} C_VEL
LIN {X 0,Y 177.052,Z 331.96,A -85,B 0,C 180,E1 -23458.933,E2 -23458.933} C_VEL
LIN {X 0,Y 174.244,Z 343.241,A -85,B 0,C 180,E1 -23461.052,E2 -23461.052} C_VEL
LIN {X 0,Y 171.635,Z 353.467,A -85,B 0,C 180,E1 -23463.557,E2 -23463.557} C_VEL
LIN {X 0,Y 168.766,Z 363.148,A -85,B 0,C 180,E1 -23466.566,E2 -23466.566} C_VEL
LIN {X 0,Y 168.69,Z 363.503,A -85,B 0,C 180,E1 -23466.693,E2 -23466.693} C_VEL
LIN {X 0,Y 167.415,Z 366.138,A -85,B 0,C 180,E1 -23467.611,E2 -23467.611} C_VEL
LIN {X 0,Y 163.541,Z 370.011,A -85,B 0,C 180,E1 -23468.973,E2 -23468.973} C_VEL
LIN {X 0,Y 159.61,Z 373.605,A -85,B 0,C 180,E1 -23470.471,E2 -23470.471} C_VEL
LIN {X 0,Y 158.293,Z 375.788,A -85,B 0,C 180,E1 -23471.585,E2 -23471.585} C_VEL
LIN {X 0,Y 156.415,Z 382.475,A -85,B 0,C 180,E1 -23475.692,E2 -23475.692} C_VEL
LIN {X 0,Y 155.41,Z 387.343,A -85,B 0,C 180,E1 -23479.578,E2 -23479.578} C_VEL
LIN {X 0,Y 154.853,Z 391.039,A -85,B 0,C 180,E1 -23483.485,E2 -23483.485} C_VEL
LIN {X 0,Y 154.776,Z 393.682,A -85,B 0,C 180,E1 -23487.397,E2 -23487.397} C_VEL
LIN {X 0,Y 154.829,Z 394.905,A -85,B 0,C 180,E1 -23490,E2 -23490} C_VEL
LIN {X 0,Y 154.699,Z 395.696,A -85,B 0,C 180,E1 -23492.604,E2 -23492.604} C_VEL
LIN {X 0,Y 154.757,Z 396.056,A -85,B 0,C 180,E1 -23495.211,E2 -23495.211} C_VEL
LIN {X 0,Y 155.44,Z 395.628,A -85,B 0,C 180,E1 -23500.42,E2 -23500.42} C_VEL
LIN {X 0,Y 156.182,Z 394.846,A -85,B 0,C 180,E1 -23503.003,E2 -23503.003} C_VEL
LIN {X 0,Y 158.452,Z 392.04,A -85,B 0,C 180,E1 -23508.088,E2 -23508.088} C_VEL
LIN {X 0,Y 161.146,Z 388.86,A -85,B 0,C 180,E1 -23511.759,E2 -23511.759} C_VEL
LIN {X 0,Y 164.358,Z 384.661,A -85,B 0,C 180,E1 -23515.316,E2 -23515.316} C_VEL
LIN {X 0,Y 168.589,Z 378.672,A -85,B 0,C 180,E1 -23519.094,E2 -23519.094} C_VEL
LIN {X 0,Y 173.409,Z 371.467,A -85,B 0,C 180,E1 -23522.48,E2 -23522.48} C_VEL
LIN {X 0,Y 177.688,Z 364.523,A -85,B 0,C 180,E1 -23524.996,E2 -23524.996} C_VEL
LIN {X 0,Y 182.323,Z 356.227,A -85,B 0,C 180,E1 -23527.382,E2 -23527.382} C_VEL
LIN {X 0,Y 186.746,Z 347.229,A -85,B 0,C 180,E1 -23529.426,E2 -23529.426} C_VEL
LIN {X 0,Y 191.459,Z 336.142,A -85,B 0,C 180,E1 -23531.357,E2 -23531.357} C_VEL
LIN {X 0,Y 195.84,Z 323.698,A -85,B 0,C 180,E1 -23532.988,E2 -23532.988} C_VEL
LIN {X 0,Y 199.278,Z 311.352,A -85,B 0,C 180,E1 -23534.15,E2 -23534.15} C_VEL
LIN {X 0,Y 202.094,Z 297.552,A -85,B 0,C 180,E1 -23535.046,E2 -23535.046} C_VEL
LIN {X 0,Y 203.717,Z 284.192,A -85,B 0,C 180,E1 -23535.614,E2 -23535.614} C_VEL
LIN {X 0,Y 206.126,Z 255.713,A -85,B 0,C 180,E1 -23536.595,E2 -23536.595} C_VEL
LIN {X 0,Y 203.057,Z 247.368,A -85,B 0,C 180,E1 -23538.577,E2 -23538.577} C_VEL
LIN {X 0,Y 199.464,Z 239.214,A -85,B 0,C 180,E1 -23541.011,E2 -23541.011} C_VEL
LIN {X 0,Y 195.507,Z 231.326,A -85,B 0,C 180,E1 -23544.072,E2 -23544.072} C_VEL
LIN {X 0,Y 192.328,Z 225.524,A -85,B 0,C 180,E1 -23546.948,E2 -23546.948} C_VEL
LIN {X 0,Y 189.431,Z 220.658,A -85,B 0,C 180,E1 -23550.077,E2 -23550.077} C_VEL
LIN {X 0,Y 186.189,Z 215.246,A -85,B 0,C 180,E1 -23554.949,E2 -23554.949} C_VEL
LIN {X 0,Y 184.948,Z 213.709,A -85,B 0,C 180,E1 -23557.666,E2 -23557.666} C_VEL
LIN {X 0,Y 183.68,Z 212.618,A -85,B 0,C 180,E1 -23563.051,E2 -23563.051} C_VEL
LIN {X 0,Y 184.331,Z 213.001,A -85,B 0,C 180,E1 -23569.01,E2 -23569.01} C_VEL
LIN {X 0,Y 186.236,Z 214.306,A -85,B 0,C 180,E1 -23573.364,E2 -23573.364} C_VEL
LIN {X 0,Y 188.497,Z 217.797,A -85,B 0,C 180,E1 -23576.948,E2 -23576.948} C_VEL
LIN {X 0,Y 189.535,Z 219.001,A -85,B 0,C 180,E1 -23578.239,E2 -23578.239} C_VEL
LIN {X 0,Y 191.9,Z 222.815,A -85,B 0,C 180,E1 -23580.847,E2 -23580.847} C_VEL
LIN {X 0,Y 193.212,Z 224.589,A -85,B 0,C 180,E1 -23582.085,E2 -23582.085} C_VEL
LIN {X 0,Y 195.56,Z 228.245,A -85,B 0,C 180,E1 -23584.122,E2 -23584.122} C_VEL
LIN {X 0,Y 199.646,Z 234.958,A -85,B 0,C 180,E1 -23587.178,E2 -23587.178} C_VEL
LIN {X 0,Y 202.968,Z 241.656,A -85,B 0,C 180,E1 -23589.406,E2 -23589.406} C_VEL
LIN {X 0,Y 206.313,Z 249.427,A -85,B 0,C 180,E1 -23591.5,E2 -23591.5} C_VEL
LIN {X 0,Y 206.579,Z 250.085,A -85,B 0,C 180,E1 -23591.661,E2 -23591.661} C_VEL
LIN {X 0,Y 203.182,Z 286.738,A -85,B 0,C 180,E1 -23592.938,E2 -23592.938} C_VEL
LIN {X 0,Y 200.884,Z 300.366,A -85,B 0,C 180,E1 -23593.736,E2 -23593.736} C_VEL
LIN {X 0,Y 198.118,Z 312.174,A -85,B 0,C 180,E1 -23594.781,E2 -23594.781} C_VEL
LIN {X 0,Y 194.429,Z 324.3,A -85,B 0,C 180,E1 -23596.254,E2 -23596.254} C_VEL
LIN {X 0,Y 190.254,Z 335.235,A -85,B 0,C 180,E1 -23597.97,E2 -23597.97} C_VEL
LIN {X 0,Y 185.974,Z 344.717,A -85,B 0,C 180,E1 -23599.884,E2 -23599.884} C_VEL
LIN {X 0,Y 181.253,Z 353.834,A -85,B 0,C 180,E1 -23602.257,E2 -23602.257} C_VEL
LIN {X 0,Y 176.61,Z 361.767,A -85,B 0,C 180,E1 -23604.915,E2 -23604.915} C_VEL
LIN {X 0,Y 171.581,Z 369.475,A -85,B 0,C 180,E1 -23608.279,E2 -23608.279} C_VEL
LIN {X 0,Y 167.976,Z 374.47,A -85,B 0,C 180,E1 -23611.105,E2 -23611.105} C_VEL
LIN {X 0,Y 163.587,Z 380.041,A -85,B 0,C 180,E1 -23615.286,E2 -23615.286} C_VEL
LIN {X 0,Y 160.037,Z 384.073,A -85,B 0,C 180,E1 -23619.779,E2 -23619.779} C_VEL
LIN {X 0,Y 157.39,Z 386.639,A -85,B 0,C 180,E1 -23624.401,E2 -23624.401} C_VEL
LIN {X 0,Y 156.061,Z 387.591,A -85,B 0,C 180,E1 -23627.506,E2 -23627.506} C_VEL
LIN {X 0,Y 155.14,Z 387.941,A -85,B 0,C 180,E1 -23630.638,E2 -23630.638} C_VEL
LIN {X 0,Y 154.379,Z 387.486,A -85,B 0,C 180,E1 -23635.029,E2 -23635.029} C_VEL
LIN {X 0,Y 154.297,Z 385.651,A -85,B 0,C 180,E1 -23639.931,E2 -23639.931} C_VEL
LIN {X 0,Y 155.021,Z 382.113,A -85,B 0,C 180,E1 -23645.056,E2 -23645.056} C_VEL
LIN {X 0,Y 155.927,Z 378.317,A -85,B 0,C 180,E1 -23648.864,E2 -23648.864} C_VEL
LIN {X 0,Y 157.37,Z 372.706,A -85,B 0,C 180,E1 -23653.125,E2 -23653.125} C_VEL
LIN {X 0,Y 159.458,Z 365.484,A -85,B 0,C 180,E1 -23657.269,E2 -23657.269} C_VEL
LIN {X 0,Y 161.804,Z 358.043,A -85,B 0,C 180,E1 -23660.604,E2 -23660.604} C_VEL
LIN {X 0,Y 164.509,Z 348.897,A -85,B 0,C 180,E1 -23663.869,E2 -23663.869} C_VEL
LIN {X 0,Y 167.349,Z 338.793,A -85,B 0,C 180,E1 -23666.69,E2 -23666.69} C_VEL
LIN {X 0,Y 170.164,Z 327.616,A -85,B 0,C 180,E1 -23669.115,E2 -23669.115} C_VEL
LIN {X 0,Y 172.811,Z 315.302,A -85,B 0,C 180,E1 -23671.165,E2 -23671.165} C_VEL
LIN {X 0,Y 174.839,Z 303.299,A -85,B 0,C 180,E1 -23672.643,E2 -23672.643} C_VEL
LIN {X 0,Y 176.612,Z 289.893,A -85,B 0,C 180,E1 -23673.795,E2 -23673.795} C_VEL
LIN {X 0,Y 177.676,Z 276.811,A -85,B 0,C 180,E1 -23674.493,E2 -23674.493} C_VEL
LIN {X 0,Y 180.333,Z 230.745,A -85,B 0,C 180,E1 -23676.344,E2 -23676.344} C_VEL
LIN {X 0,Y 174.948,Z 215.616,A -85,B 0,C 180,E1 -23678.196,E2 -23678.196} C_VEL
LIN {X 0,Y 164.094,Z 195.322,A -85,B 0,C 180,E1 -23681.786,E2 -23681.786} C_VEL
LIN {X 0,Y 159.971,Z 188.685,A -85,B 0,C 180,E1 -23683.239,E2 -23683.239} C_VEL
LIN {X 0,Y 157.921,Z 185.627,A -85,B 0,C 180,E1 -23683.985,E2 -23683.985} C_VEL
LIN {X 0,Y 157.449,Z 183.872,A -85,B 0,C 180,E1 -23684.295,E2 -23684.295} C_VEL
LIN {X 0,Y 157.362,Z 183.885,A -85,B 0,C 180,E1 -23690.299,E2 -23690.299} C_VEL
LIN {X 0,Y 157.267,Z 183.889,A -85,B 0,C 180,E1 -23696.649,E2 -23696.649} C_VEL
LIN {X 0,Y 157.266,Z 183.867,A -85,B 0,C 180,E1 -23702.43,E2 -23702.43} C_VEL
LIN {X 0,Y 157.268,Z 183.881,A -85,B 0,C 180,E1 -23706.448,E2 -23706.448} C_VEL
LIN {X 0,Y 157.191,Z 183.894,A -85,B 0,C 180,E1 -23712.117,E2 -23712.117} C_VEL
LIN {X 0,Y 157.19,Z 183.861,A -85,B 0,C 180,E1 -23717.882,E2 -23717.882} C_VEL
LIN {X 0,Y 157.26,Z 183.896,A -85,B 0,C 180,E1 -23723.556,E2 -23723.556} C_VEL
LIN {X 0,Y 157.281,Z 183.878,A -85,B 0,C 180,E1 -23728.104,E2 -23728.104} C_VEL
LIN {X 0,Y 157.311,Z 183.887,A -85,B 0,C 180,E1 -23733.464,E2 -23733.464} C_VEL
LIN {X 0,Y 157.361,Z 183.881,A -85,B 0,C 180,E1 -23739.702,E2 -23739.702} C_VEL
LIN {X 0,Y 157.409,Z 183.863,A -85,B 0,C 180,E1 -23744.461,E2 -23744.461} C_VEL
LIN {X 0,Y 157.689,Z 183.842,A -85,B 0,C 180,E1 -23749.731,E2 -23749.731} C_VEL
LIN {X 0,Y 157.762,Z 183.825,A -85,B 0,C 180,E1 -23752.32,E2 -23752.32} C_VEL
LIN {X 0,Y 158.238,Z 183.772,A -85,B 0,C 180,E1 -23760,E2 -23760} C_VEL
LIN {X 0,Y 157.759,Z 183.784,A -85,B 0,C 180,E1 -23767.68,E2 -23767.68} C_VEL
LIN {X 0,Y 157.632,Z 183.84,A -85,B 0,C 180,E1 -23771.223,E2 -23771.223} C_VEL
LIN {X 0,Y 157.406,Z 183.874,A -85,B 0,C 180,E1 -23775.539,E2 -23775.539} C_VEL
LIN {X 0,Y 157.308,Z 183.853,A -85,B 0,C 180,E1 -23780.941,E2 -23780.941} C_VEL
LIN {X 0,Y 157.311,Z 183.889,A -85,B 0,C 180,E1 -23786.681,E2 -23786.681} C_VEL
LIN {X 0,Y 157.269,Z 183.896,A -85,B 0,C 180,E1 -23792.429,E2 -23792.429} C_VEL
LIN {X 0,Y 157.259,Z 183.899,A -85,B 0,C 180,E1 -23796.444,E2 -23796.444} C_VEL
LIN {X 0,Y 157.191,Z 183.903,A -85,B 0,C 180,E1 -23802.117,E2 -23802.117} C_VEL
LIN {X 0,Y 157.245,Z 183.961,A -85,B 0,C 180,E1 -23803.298,E2 -23803.298} C_VEL
LIN {X 0,Y 158.287,Z 186.802,A -85,B 0,C 180,E1 -23803.767,E2 -23803.767} C_VEL
LIN {X 0,Y 159.982,Z 189.276,A -85,B 0,C 180,E1 -23804.38,E2 -23804.38} C_VEL
LIN {X 0,Y 167.638,Z 205.08,A -85,B 0,C 180,E1 -23807.211,E2 -23807.211} C_VEL
LIN {X 0,Y 174.106,Z 220.912,A -85,B 0,C 180,E1 -23809.502,E2 -23809.502} C_VEL
LIN {X 0,Y 178.621,Z 233.831,A -85,B 0,C 180,E1 -23811.078,E2 -23811.078} C_VEL
LIN {X 0,Y 179.734,Z 245.685,A -85,B 0,C 180,E1 -23811.89,E2 -23811.89} C_VEL
LIN {X 0,Y 176.866,Z 293.194,A -85,B 0,C 180,E1 -23813.854,E2 -23813.854} C_VEL
LIN {X 0,Y 175.196,Z 307.328,A -85,B 0,C 180,E1 -23814.872,E2 -23814.872} C_VEL
LIN {X 0,Y 173.284,Z 318.911,A -85,B 0,C 180,E1 -23816.105,E2 -23816.105} C_VEL
LIN {X 0,Y 171.002,Z 330.03,A -85,B 0,C 180,E1 -23817.704,E2 -23817.704} C_VEL
LIN {X 0,Y 167.969,Z 341.59,A -85,B 0,C 180,E1 -23819.861,E2 -23819.861} C_VEL
LIN {X 0,Y 165.211,Z 352.113,A -85,B 0,C 180,E1 -23822.444,E2 -23822.444} C_VEL
LIN {X 0,Y 162.76,Z 360.608,A -85,B 0,C 180,E1 -23825.065,E2 -23825.065} C_VEL
LIN {X 0,Y 160.442,Z 368.621,A -85,B 0,C 180,E1 -23828.14,E2 -23828.14} C_VEL
LIN {X 0,Y 158.293,Z 375.788,A -85,B 0,C 180,E1 -23831.585,E2 -23831.585} C_VEL
LIN {X 0,Y 156.783,Z 378.902,A -85,B 0,C 180,E1 -23833.337,E2 -23833.337} C_VEL
LIN {X 0,Y 152.747,Z 383.367,A -85,B 0,C 180,E1 -23836.26,E2 -23836.26} C_VEL
LIN {X 0,Y 148.997,Z 387.15,A -85,B 0,C 180,E1 -23839.449,E2 -23839.449} C_VEL
LIN {X 0,Y 147.978,Z 389.176,A -85,B 0,C 180,E1 -23841.558,E2 -23841.558} C_VEL
LIN {X 0,Y 147.706,Z 391.588,A -85,B 0,C 180,E1 -23844.539,E2 -23844.539} C_VEL
LIN {X 0,Y 147.689,Z 393.603,A -85,B 0,C 180,E1 -23847.887,E2 -23847.887} C_VEL
LIN {X 0,Y 147.635,Z 395.046,A -85,B 0,C 180,E1 -23851.448,E2 -23851.448} C_VEL
LIN {X 0,Y 147.688,Z 395.836,A -85,B 0,C 180,E1 -23855.461,E2 -23855.461} C_VEL
LIN {X 0,Y 148.429,Z 395.503,A -85,B 0,C 180,E1 -23860.918,E2 -23860.918} C_VEL
LIN {X 0,Y 150.306,Z 393.664,A -85,B 0,C 180,E1 -23866.293,E2 -23866.293} C_VEL
LIN {X 0,Y 151.709,Z 392.12,A -85,B 0,C 180,E1 -23868.922,E2 -23868.922} C_VEL
LIN {X 0,Y 154.575,Z 389.047,A -85,B 0,C 180,E1 -23872.735,E2 -23872.735} C_VEL
LIN {X 0,Y 157.969,Z 384.96,A -85,B 0,C 180,E1 -23876.417,E2 -23876.417} C_VEL
LIN {X 0,Y 162.695,Z 378.774,A -85,B 0,C 180,E1 -23880.502,E2 -23880.502} C_VEL
LIN {X 0,Y 167.503,Z 372.087,A -85,B 0,C 180,E1 -23883.776,E2 -23883.776} C_VEL
LIN {X 0,Y 171.969,Z 365.317,A -85,B 0,C 180,E1 -23886.341,E2 -23886.341} C_VEL
LIN {X 0,Y 177.766,Z 355.438,A -85,B 0,C 180,E1 -23889.24,E2 -23889.24} C_VEL
LIN {X 0,Y 182.987,Z 345.133,A -85,B 0,C 180,E1 -23891.493,E2 -23891.493} C_VEL
LIN {X 0,Y 187.964,Z 333.63,A -85,B 0,C 180,E1 -23893.397,E2 -23893.397} C_VEL
LIN {X 0,Y 191.954,Z 322.345,A -85,B 0,C 180,E1 -23894.814,E2 -23894.814} C_VEL
LIN {X 0,Y 195.249,Z 310.861,A -85,B 0,C 180,E1 -23895.862,E2 -23895.862} C_VEL
LIN {X 0,Y 198.21,Z 296.83,A -85,B 0,C 180,E1 -23896.756,E2 -23896.756} C_VEL
LIN {X 0,Y 199.983,Z 282.324,A -85,B 0,C 180,E1 -23897.344,E2 -23897.344} C_VEL
LIN {X 0,Y 202.111,Z 258.466,A -85,B 0,C 180,E1 -23898.17,E2 -23898.17} C_VEL
LIN {X 0,Y 198.877,Z 249.74,A -85,B 0,C 180,E1 -23900.437,E2 -23900.437} C_VEL
LIN {X 0,Y 195.923,Z 243.055,A -85,B 0,C 180,E1 -23902.69,E2 -23902.69} C_VEL
LIN {X 0,Y 192.98,Z 236.821,A -85,B 0,C 180,E1 -23905.183,E2 -23905.183} C_VEL
LIN {X 0,Y 190.285,Z 231.677,A -85,B 0,C 180,E1 -23907.853,E2 -23907.853} C_VEL
LIN {X 0,Y 187.721,Z 227.079,A -85,B 0,C 180,E1 -23910.876,E2 -23910.876} C_VEL
LIN {X 0,Y 184.871,Z 222.032,A -85,B 0,C 180,E1 -23915.52,E2 -23915.52} C_VEL
LIN {X 0,Y 183.74,Z 220.602,A -85,B 0,C 180,E1 -23918.178,E2 -23918.178} C_VEL
LIN {X 0,Y 182.631,Z 219.551,A -85,B 0,C 180,E1 -23924.167,E2 -23924.167} C_VEL
LIN {X 0,Y 183.831,Z 220.364,A -85,B 0,C 180,E1 -23930.427,E2 -23930.427} C_VEL
LIN {X 0,Y 184.977,Z 221.174,A -85,B 0,C 180,E1 -23932.907,E2 -23932.907} C_VEL
LIN {X 0,Y 187.009,Z 224.53,A -85,B 0,C 180,E1 -23936.372,E2 -23936.372} C_VEL
LIN {X 0,Y 187.968,Z 225.678,A -85,B 0,C 180,E1 -23937.628,E2 -23937.628} C_VEL
LIN {X 0,Y 190.248,Z 229.479,A -85,B 0,C 180,E1 -23940.305,E2 -23940.305} C_VEL
LIN {X 0,Y 191.592,Z 231.508,A -85,B 0,C 180,E1 -23941.642,E2 -23941.642} C_VEL
LIN {X 0,Y 193.533,Z 234.712,A -85,B 0,C 180,E1 -23943.441,E2 -23943.441} C_VEL
LIN {X 0,Y 197.25,Z 241.111,A -85,B 0,C 180,E1 -23946.374,E2 -23946.374} C_VEL
LIN {X 0,Y 200.912,Z 249.071,A -85,B 0,C 180,E1 -23948.995,E2 -23948.995} C_VEL
LIN {X 0,Y 202.52,Z 252.904,A -85,B 0,C 180,E1 -23950.059,E2 -23950.059} C_VEL
LIN {X 0,Y 199.369,Z 286.04,A -85,B 0,C 180,E1 -23951.222,E2 -23951.222} C_VEL
LIN {X 0,Y 197.051,Z 299.568,A -85,B 0,C 180,E1 -23951.994,E2 -23951.994} C_VEL
LIN {X 0,Y 194.278,Z 311.12,A -85,B 0,C 180,E1 -23952.974,E2 -23952.974} C_VEL
LIN {X 0,Y 190.485,Z 323.353,A -85,B 0,C 180,E1 -23954.417,E2 -23954.417} C_VEL
LIN {X 0,Y 185.775,Z 335.278,A -85,B 0,C 180,E1 -23956.268,E2 -23956.268} C_VEL
LIN {X 0,Y 180.734,Z 345.887,A -85,B 0,C 180,E1 -23958.438,E2 -23958.438} C_VEL
LIN {X 0,Y 175.16,Z 355.899,A -85,B 0,C 180,E1 -23961.169,E2 -23961.169} C_VEL
LIN {X 0,Y 169.661,Z 364.562,A -85,B 0,C 180,E1 -23964.31,E2 -23964.31} C_VEL
LIN {X 0,Y 165.639,Z 370.25,A -85,B 0,C 180,E1 -23966.997,E2 -23966.997} C_VEL
LIN {X 0,Y 160.581,Z 376.624,A -85,B 0,C 180,E1 -23970.944,E2 -23970.944} C_VEL
LIN {X 0,Y 155.799,Z 382.031,A -85,B 0,C 180,E1 -23975.711,E2 -23975.711} C_VEL
LIN {X 0,Y 152.506,Z 385.331,A -85,B 0,C 180,E1 -23980.178,E2 -23980.178} C_VEL
LIN {X 0,Y 149.805,Z 387.472,A -85,B 0,C 180,E1 -23985.273,E2 -23985.273} C_VEL
LIN {X 0,Y 148.375,Z 388.121,A -85,B 0,C 180,E1 -23989.276,E2 -23989.276} C_VEL
LIN {X 0,Y 147.393,Z 387.75,A -85,B 0,C 180,E1 -23994.155,E2 -23994.155} C_VEL
LIN {X 0,Y 147.148,Z 386.024,A -85,B 0,C 180,E1 -23999.284,E2 -23999.284} C_VEL
LIN {X 0,Y 147.553,Z 383.765,A -85,B 0,C 180,E1 -24003.098,E2 -24003.098} C_VEL
LIN {X 0,Y 148.556,Z 379.832,A -85,B 0,C 180,E1 -24007.761,E2 -24007.761} C_VEL
LIN {X 0,Y 149.844,Z 374.576,A -85,B 0,C 180,E1 -24012.25,E2 -24012.25} C_VEL
LIN {X 0,Y 151.887,Z 367.801,A -85,B 0,C 180,E1 -24016.623,E2 -24016.623} C_VEL
LIN {X 0,Y 154.144,Z 360.793,A -85,B 0,C 180,E1 -24020.155,E2 -24020.155} C_VEL
LIN {X 0,Y 156.792,Z 352.295,A -85,B 0,C 180,E1 -24023.566,E2 -24023.566} C_VEL
LIN {X 0,Y 159.638,Z 342.876,A -85,B 0,C 180,E1 -24026.529,E2 -24026.529} C_VEL
LIN {X 0,Y 162.693,Z 331.732,A -85,B 0,C 180,E1 -24029.276,E2 -24029.276} C_VEL
LIN {X 0,Y 165.507,Z 319.827,A -85,B 0,C 180,E1 -24031.521,E2 -24031.521} C_VEL
LIN {X 0,Y 167.853,Z 307.464,A -85,B 0,C 180,E1 -24033.269,E2 -24033.269} C_VEL
LIN {X 0,Y 169.77,Z 294.684,A -85,B 0,C 180,E1 -24034.565,E2 -24034.565} C_VEL
LIN {X 0,Y 171.181,Z 281.579,A -85,B 0,C 180,E1 -24035.404,E2 -24035.404} C_VEL
LIN {X 0,Y 174.148,Z 232.384,A -85,B 0,C 180,E1 -24037.465,E2 -24037.465} C_VEL
LIN {X 0,Y 169.608,Z 219.325,A -85,B 0,C 180,E1 -24039.141,E2 -24039.141} C_VEL
LIN {X 0,Y 159.396,Z 200.006,A -85,B 0,C 180,E1 -24042.696,E2 -24042.696} C_VEL
LIN {X 0,Y 152.366,Z 188.85,A -85,B 0,C 180,E1 -24045.374,E2 -24045.374} C_VEL
LIN {X 0,Y 150.744,Z 186.363,A -85,B 0,C 180,E1 -24046.022,E2 -24046.022} C_VEL
LIN {X 0,Y 150.32,Z 184.744,A -85,B 0,C 180,E1 -24046.291,E2 -24046.291} C_VEL
LIN {X 0,Y 150.285,Z 184.766,A -85,B 0,C 180,E1 -24050.724,E2 -24050.724} C_VEL
LIN {X 0,Y 150.186,Z 184.774,A -85,B 0,C 180,E1 -24057.237,E2 -24057.237} C_VEL
LIN {X 0,Y 150.206,Z 184.743,A -85,B 0,C 180,E1 -24062.626,E2 -24062.626} C_VEL
LIN {X 0,Y 150.173,Z 184.772,A -85,B 0,C 180,E1 -24067.474,E2 -24067.474} C_VEL
LIN {X 0,Y 150.135,Z 184.776,A -85,B 0,C 180,E1 -24071.498,E2 -24071.498} C_VEL
LIN {X 0,Y 150.126,Z 184.736,A -85,B 0,C 180,E1 -24075.395,E2 -24075.395} C_VEL
LIN {X 0,Y 150.137,Z 184.752,A -85,B 0,C 180,E1 -24079.054,E2 -24079.054} C_VEL
LIN {X 0,Y 150.176,Z 184.776,A -85,B 0,C 180,E1 -24082.71,E2 -24082.71} C_VEL
LIN {X 0,Y 150.206,Z 184.76,A -85,B 0,C 180,E1 -24087.374,E2 -24087.374} C_VEL
LIN {X 0,Y 150.24,Z 184.771,A -85,B 0,C 180,E1 -24092.723,E2 -24092.723} C_VEL
LIN {X 0,Y 150.286,Z 184.761,A -85,B 0,C 180,E1 -24099.276,E2 -24099.276} C_VEL
LIN {X 0,Y 150.314,Z 184.752,A -85,B 0,C 180,E1 -24103.708,E2 -24103.708} C_VEL
LIN {X 0,Y 150.609,Z 184.724,A -85,B 0,C 180,E1 -24109.242,E2 -24109.242} C_VEL
LIN {X 0,Y 150.7,Z 184.707,A -85,B 0,C 180,E1 -24111.957,E2 -24111.957} C_VEL
LIN {X 0,Y 151.199,Z 184.648,A -85,B 0,C 180,E1 -24120,E2 -24120} C_VEL
LIN {X 0,Y 150.682,Z 184.666,A -85,B 0,C 180,E1 -24128.043,E2 -24128.043} C_VEL
LIN {X 0,Y 150.574,Z 184.72,A -85,B 0,C 180,E1 -24131.427,E2 -24131.427} C_VEL
LIN {X 0,Y 150.312,Z 184.754,A -85,B 0,C 180,E1 -24136.292,E2 -24136.292} C_VEL
LIN {X 0,Y 150.284,Z 184.726,A -85,B 0,C 180,E1 -24140.723,E2 -24140.723} C_VEL
LIN {X 0,Y 150.24,Z 184.767,A -85,B 0,C 180,E1 -24147.277,E2 -24147.277} C_VEL
LIN {X 0,Y 150.209,Z 184.774,A -85,B 0,C 180,E1 -24152.628,E2 -24152.628} C_VEL
LIN {X 0,Y 150.17,Z 184.781,A -85,B 0,C 180,E1 -24157.474,E2 -24157.474} C_VEL
LIN {X 0,Y 150.137,Z 184.779,A -85,B 0,C 180,E1 -24161.28,E2 -24161.28} C_VEL
LIN {X 0,Y 151.171,Z 187.681,A -85,B 0,C 180,E1 -24161.791,E2 -24161.791} C_VEL
LIN {X 0,Y 152.878,Z 189.997,A -85,B 0,C 180,E1 -24162.445,E2 -24162.445} C_VEL
LIN {X 0,Y 155.549,Z 194.561,A -85,B 0,C 180,E1 -24163.501,E2 -24163.501} C_VEL
LIN {X 0,Y 162.638,Z 209.352,A -85,B 0,C 180,E1 -24166.268,E2 -24166.268} C_VEL
LIN {X 0,Y 169.179,Z 225.761,A -85,B 0,C 180,E1 -24168.716,E2 -24168.716} C_VEL
LIN {X 0,Y 172.713,Z 236.364,A -85,B 0,C 180,E1 -24170.046,E2 -24170.046} C_VEL
LIN {X 0,Y 173.582,Z 246.32,A -85,B 0,C 180,E1 -24170.753,E2 -24170.753} C_VEL
LIN {X 0,Y 170.605,Z 293.464,A -85,B 0,C 180,E1 -24172.767,E2 -24172.767} C_VEL
LIN {X 0,Y 168.871,Z 307.445,A -85,B 0,C 180,E1 -24173.811,E2 -24173.811} C_VEL
LIN {X 0,Y 166.761,Z 319.442,A -85,B 0,C 180,E1 -24175.139,E2 -24175.139} C_VEL
LIN {X 0,Y 164.196,Z 331.175,A -85,B 0,C 180,E1 -24176.925,E2 -24176.925} C_VEL
LIN {X 0,Y 161.144,Z 342.513,A -85,B 0,C 180,E1 -24179.172,E2 -24179.172} C_VEL
LIN {X 0,Y 158.326,Z 352.825,A -85,B 0,C 180,E1 -24181.859,E2 -24181.859} C_VEL
LIN {X 0,Y 155.466,Z 361.835,A -85,B 0,C 180,E1 -24184.829,E2 -24184.829} C_VEL
LIN {X 0,Y 153.345,Z 369.016,A -85,B 0,C 180,E1 -24187.783,E2 -24187.783} C_VEL
LIN {X 0,Y 150.999,Z 376.604,A -85,B 0,C 180,E1 -24191.689,E2 -24191.689} C_VEL
LIN {X 0,Y 149.055,Z 383.579,A -85,B 0,C 180,E1 -24196.364,E2 -24196.364} C_VEL
LIN {X 0,Y 148.148,Z 388.151,A -85,B 0,C 180,E1 -24200.443,E2 -24200.443} C_VEL
LIN {X 0,Y 147.978,Z 389.176,A -85,B 0,C 180,E1 -24201.558,E2 -24201.558} C_VEL
LIN {X 0,Y 147.098,Z 390.985,A -85,B 0,C 180,E1 -24203.717,E2 -24203.717} C_VEL
LIN {X 0,Y 145.401,Z 392.444,A -85,B 0,C 180,E1 -24205.879,E2 -24205.879} C_VEL
LIN {X 0,Y 141.633,Z 394.433,A -85,B 0,C 180,E1 -24210.374,E2 -24210.374} C_VEL
LIN {X 0,Y 140.603,Z 395.056,A -85,B 0,C 180,E1 -24212.767,E2 -24212.767} C_VEL
LIN {X 0,Y 140.522,Z 395.206,A -85,B 0,C 180,E1 -24213.581,E2 -24213.581} C_VEL
LIN {X 0,Y 140.883,Z 395.685,A -85,B 0,C 180,E1 -24218.607,E2 -24218.607} C_VEL
LIN {X 0,Y 142.309,Z 394.701,A -85,B 0,C 180,E1 -24224.296,E2 -24224.296} C_VEL
LIN {X 0,Y 145.003,Z 392.198,A -85,B 0,C 180,E1 -24229.833,E2 -24229.833} C_VEL
LIN {X 0,Y 148.053,Z 389.228,A -85,B 0,C 180,E1 -24233.797,E2 -24233.797} C_VEL
LIN {X 0,Y 151.647,Z 385.265,A -85,B 0,C 180,E1 -24237.61,E2 -24237.61} C_VEL
LIN {X 0,Y 155.853,Z 380.223,A -85,B 0,C 180,E1 -24241.236,E2 -24241.236} C_VEL
LIN {X 0,Y 160.766,Z 373.935,A -85,B 0,C 180,E1 -24244.633,E2 -24244.633} C_VEL
LIN {X 0,Y 166.352,Z 366.112,A -85,B 0,C 180,E1 -24247.778,E2 -24247.778} C_VEL
LIN {X 0,Y 172.387,Z 356.47,A -85,B 0,C 180,E1 -24250.716,E2 -24250.716} C_VEL
LIN {X 0,Y 177.808,Z 346.565,A -85,B 0,C 180,E1 -24252.986,E2 -24252.986} C_VEL
LIN {X 0,Y 182.95,Z 335.459,A -85,B 0,C 180,E1 -24254.901,E2 -24254.901} C_VEL
LIN {X 0,Y 187.093,Z 324.71,A -85,B 0,C 180,E1 -24256.313,E2 -24256.313} C_VEL
LIN {X 0,Y 190.776,Z 312.957,A -85,B 0,C 180,E1 -24257.459,E2 -24257.459} C_VEL
LIN {X 0,Y 193.847,Z 299.94,A -85,B 0,C 180,E1 -24258.334,E2 -24258.334} C_VEL
LIN {X 0,Y 195.895,Z 286.004,A -85,B 0,C 180,E1 -24258.974,E2 -24258.974} C_VEL
LIN {X 0,Y 198.223,Z 261.265,A -85,B 0,C 180,E1 -24259.824,E2 -24259.824} C_VEL
LIN {X 0,Y 195.293,Z 253.102,A -85,B 0,C 180,E1 -24262.131,E2 -24262.131} C_VEL
LIN {X 0,Y 191.704,Z 244.918,A -85,B 0,C 180,E1 -24265.213,E2 -24265.213} C_VEL
LIN {X 0,Y 188.648,Z 238.388,A -85,B 0,C 180,E1 -24268.391,E2 -24268.391} C_VEL
LIN {X 0,Y 186.116,Z 233.596,A -85,B 0,C 180,E1 -24271.595,E2 -24271.595} C_VEL
LIN {X 0,Y 183.603,Z 228.818,A -85,B 0,C 180,E1 -24276.044,E2 -24276.044} C_VEL
LIN {X 0,Y 182.781,Z 227.689,A -85,B 0,C 180,E1 -24278.057,E2 -24278.057} C_VEL
LIN {X 0,Y 181.704,Z 226.665,A -85,B 0,C 180,E1 -24282.933,E2 -24282.933} C_VEL
LIN {X 0,Y 182.305,Z 227.022,A -85,B 0,C 180,E1 -24288.887,E2 -24288.887} C_VEL
LIN {X 0,Y 183.74,Z 228.033,A -85,B 0,C 180,E1 -24292.459,E2 -24292.459} C_VEL
LIN {X 0,Y 185.763,Z 231.46,A -85,B 0,C 180,E1 -24296.092,E2 -24296.092} C_VEL
LIN {X 0,Y 186.511,Z 232.606,A -85,B 0,C 180,E1 -24297.147,E2 -24297.147} C_VEL
LIN {X 0,Y 189.554,Z 237.643,A -85,B 0,C 180,E1 -24300.747,E2 -24300.747} C_VEL
LIN {X 0,Y 191.716,Z 241.369,A -85,B 0,C 180,E1 -24302.864,E2 -24302.864} C_VEL
LIN {X 0,Y 195.157,Z 247.712,A -85,B 0,C 180,E1 -24305.752,E2 -24305.752} C_VEL
LIN {X 0,Y 198.621,Z 256.068,A -85,B 0,C 180,E1 -24308.421,E2 -24308.421} C_VEL
LIN {X 0,Y 195.5,Z 287.016,A -85,B 0,C 180,E1 -24309.509,E2 -24309.509} C_VEL
LIN {X 0,Y 192.995,Z 300.858,A -85,B 0,C 180,E1 -24310.318,E2 -24310.318} C_VEL
LIN {X 0,Y 189.957,Z 312.671,A -85,B 0,C 180,E1 -24311.348,E2 -24311.348} C_VEL
LIN {X 0,Y 186.391,Z 323.548,A -85,B 0,C 180,E1 -24312.642,E2 -24312.642} C_VEL
LIN {X 0,Y 181.471,Z 335.478,A -85,B 0,C 180,E1 -24314.486,E2 -24314.486} C_VEL
LIN {X 0,Y 177.017,Z 344.533,A -85,B 0,C 180,E1 -24316.31,E2 -24316.31} C_VEL
LIN {X 0,Y 171.645,Z 353.989,A -85,B 0,C 180,E1 -24318.762,E2 -24318.762} C_VEL
LIN {X 0,Y 166.247,Z 362.222,A -85,B 0,C 180,E1 -24321.558,E2 -24321.558} C_VEL
LIN {X 0,Y 160.996,Z 369.424,A -85,B 0,C 180,E1 -24324.78,E2 -24324.78} C_VEL
LIN {X 0,Y 155.901,Z 375.63,A -85,B 0,C 180,E1 -24328.47,E2 -24328.47} C_VEL
LIN {X 0,Y 150.844,Z 381.059,A -85,B 0,C 180,E1 -24333.002,E2 -24333.002} C_VEL
LIN {X 0,Y 148.041,Z 383.797,A -85,B 0,C 180,E1 -24336.191,E2 -24336.191} C_VEL
LIN {X 0,Y 145.668,Z 385.837,A -85,B 0,C 180,E1 -24339.47,E2 -24339.47} C_VEL
LIN {X 0,Y 143.512,Z 387.43,A -85,B 0,C 180,E1 -24343.283,E2 -24343.283} C_VEL
LIN {X 0,Y 141.582,Z 388.315,A -85,B 0,C 180,E1 -24348.124,E2 -24348.124} C_VEL
LIN {X 0,Y 140.404,Z 388.007,A -85,B 0,C 180,E1 -24353.216,E2 -24353.216} C_VEL
LIN {X 0,Y 140.054,Z 386.369,A -85,B 0,C 180,E1 -24358.548,E2 -24358.548} C_VEL
LIN {X 0,Y 140.601,Z 383.116,A -85,B 0,C 180,E1 -24364.125,E2 -24364.125} C_VEL
LIN {X 0,Y 141.527,Z 379.717,A -85,B 0,C 180,E1 -24368.134,E2 -24368.134} C_VEL
LIN {X 0,Y 142.892,Z 374.372,A -85,B 0,C 180,E1 -24372.836,E2 -24372.836} C_VEL
LIN {X 0,Y 145.079,Z 367.453,A -85,B 0,C 180,E1 -24377.444,E2 -24377.444} C_VEL
LIN {X 0,Y 147.477,Z 360.402,A -85,B 0,C 180,E1 -24381.09,E2 -24381.09} C_VEL
LIN {X 0,Y 150.272,Z 351.739,A -85,B 0,C 180,E1 -24384.633,E2 -24384.633} C_VEL
LIN {X 0,Y 153.385,Z 341.759,A -85,B 0,C 180,E1 -24387.821,E2 -24387.821} C_VEL
LIN {X 0,Y 156.603,Z 330.352,A -85,B 0,C 180,E1 -24390.643,E2 -24390.643} C_VEL
LIN {X 0,Y 159.42,Z 318.607,A -85,B 0,C 180,E1 -24392.843,E2 -24392.843} C_VEL
LIN {X 0,Y 161.809,Z 306.43,A -85,B 0,C 180,E1 -24394.563,E2 -24394.563} C_VEL
LIN {X 0,Y 163.795,Z 293.21,A -85,B 0,C 180,E1 -24395.873,E2 -24395.873} C_VEL
LIN {X 0,Y 165.207,Z 279.18,A -85,B 0,C 180,E1 -24396.74,E2 -24396.74} C_VEL
LIN {X 0,Y 168.054,Z 234.115,A -85,B 0,C 180,E1 -24398.658,E2 -24398.658} C_VEL
LIN {X 0,Y 164.09,Z 222.629,A -85,B 0,C 180,E1 -24400.193,E2 -24400.193} C_VEL
LIN {X 0,Y 154.492,Z 204.296,A -85,B 0,C 180,E1 -24403.755,E2 -24403.755} C_VEL
LIN {X 0,Y 147.591,Z 193.34,A -85,B 0,C 180,E1 -24406.517,E2 -24406.517} C_VEL
LIN {X 0,Y 145.5,Z 189.976,A -85,B 0,C 180,E1 -24407.425,E2 -24407.425} C_VEL
LIN {X 0,Y 143.752,Z 187.556,A -85,B 0,C 180,E1 -24408.182,E2 -24408.182} C_VEL
LIN {X 0,Y 143.236,Z 185.634,A -85,B 0,C 180,E1 -24408.545,E2 -24408.545} C_VEL
LIN {X 0,Y 143.105,Z 185.638,A -85,B 0,C 180,E1 -24413.134,E2 -24413.134} C_VEL
LIN {X 0,Y 143.143,Z 185.655,A -85,B 0,C 180,E1 -24417.9,E2 -24417.9} C_VEL
LIN {X 0,Y 143.138,Z 185.619,A -85,B 0,C 180,E1 -24423.415,E2 -24423.415} C_VEL
LIN {X 0,Y 143.055,Z 185.666,A -85,B 0,C 180,E1 -24429.693,E2 -24429.693} C_VEL
LIN {X 0,Y 143.034,Z 185.637,A -85,B 0,C 180,E1 -24433.464,E2 -24433.464} C_VEL
LIN {X 0,Y 143.037,Z 185.617,A -85,B 0,C 180,E1 -24437.478,E2 -24437.478} C_VEL
LIN {X 0,Y 143.073,Z 185.657,A -85,B 0,C 180,E1 -24441.809,E2 -24441.809} C_VEL
LIN {X 0,Y 143.174,Z 185.635,A -85,B 0,C 180,E1 -24447.319,E2 -24447.319} C_VEL
LIN {X 0,Y 143.184,Z 185.649,A -85,B 0,C 180,E1 -24452.069,E2 -24452.069} C_VEL
LIN {X 0,Y 143.224,Z 185.637,A -85,B 0,C 180,E1 -24458.802,E2 -24458.802} C_VEL
LIN {X 0,Y 143.254,Z 185.635,A -85,B 0,C 180,E1 -24462.881,E2 -24462.881} C_VEL
LIN {X 0,Y 143.535,Z 185.604,A -85,B 0,C 180,E1 -24468.705,E2 -24468.705} C_VEL
LIN {X 0,Y 143.622,Z 185.592,A -85,B 0,C 180,E1 -24471.558,E2 -24471.558} C_VEL
LIN {X 0,Y 144.157,Z 185.525,A -85,B 0,C 180,E1 -24480,E2 -24480} C_VEL
LIN {X 0,Y 143.608,Z 185.549,A -85,B 0,C 180,E1 -24488.442,E2 -24488.442} C_VEL
LIN {X 0,Y 143.499,Z 185.601,A -85,B 0,C 180,E1 -24491.613,E2 -24491.613} C_VEL
LIN {X 0,Y 143.252,Z 185.624,A -85,B 0,C 180,E1 -24497.119,E2 -24497.119} C_VEL
LIN {X 0,Y 143.222,Z 185.606,A -85,B 0,C 180,E1 -24501.196,E2 -24501.196} C_VEL
LIN {X 0,Y 143.183,Z 185.642,A -85,B 0,C 180,E1 -24507.93,E2 -24507.93} C_VEL
LIN {X 0,Y 143.139,Z 185.651,A -85,B 0,C 180,E1 -24513.416,E2 -24513.416} C_VEL
LIN {X 0,Y 143.055,Z 185.692,A -85,B 0,C 180,E1 -24519.036,E2 -24519.036} C_VEL
LIN {X 0,Y 144.06,Z 188.516,A -85,B 0,C 180,E1 -24519.588,E2 -24519.588} C_VEL
LIN {X 0,Y 145.858,Z 190.84,A -85,B 0,C 180,E1 -24520.351,E2 -24520.351} C_VEL
LIN {X 0,Y 150.962,Z 199.314,A -85,B 0,C 180,E1 -24522.503,E2 -24522.503} C_VEL
LIN {X 0,Y 157.385,Z 213.054,A -85,B 0,C 180,E1 -24525.168,E2 -24525.168} C_VEL
LIN {X 0,Y 163.537,Z 228.674,A -85,B 0,C 180,E1 -24527.615,E2 -24527.615} C_VEL
LIN {X 0,Y 166.874,Z 238.985,A -85,B 0,C 180,E1 -24528.95,E2 -24528.95} C_VEL
LIN {X 0,Y 167.479,Z 247.197,A -85,B 0,C 180,E1 -24529.543,E2 -24529.543} C_VEL
LIN {X 0,Y 164.488,Z 292.625,A -85,B 0,C 180,E1 -24531.522,E2 -24531.522} C_VEL
LIN {X 0,Y 162.819,Z 306.073,A -85,B 0,C 180,E1 -24532.529,E2 -24532.529} C_VEL
LIN {X 0,Y 160.523,Z 318.951,A -85,B 0,C 180,E1 -24533.962,E2 -24533.962} C_VEL
LIN {X 0,Y 157.854,Z 330.749,A -85,B 0,C 180,E1 -24535.799,E2 -24535.799} C_VEL
LIN {X 0,Y 154.665,Z 342.124,A -85,B 0,C 180,E1 -24538.113,E2 -24538.113} C_VEL
LIN {X 0,Y 152.016,Z 351.413,A -85,B 0,C 180,E1 -24540.579,E2 -24540.579} C_VEL
LIN {X 0,Y 149.326,Z 359.986,A -85,B 0,C 180,E1 -24543.41,E2 -24543.41} C_VEL
LIN {X 0,Y 146.778,Z 368.027,A -85,B 0,C 180,E1 -24546.732,E2 -24546.732} C_VEL
LIN {X 0,Y 144.247,Z 375.758,A -85,B 0,C 180,E1 -24550.799,E2 -24550.799} C_VEL
LIN {X 0,Y 142.602,Z 381.027,A -85,B 0,C 180,E1 -24554.272,E2 -24554.272} C_VEL
LIN {X 0,Y 141.391,Z 386.119,A -85,B 0,C 180,E1 -24558.532,E2 -24558.532} C_VEL
LIN {X 0,Y 140.737,Z 390.026,A -85,B 0,C 180,E1 -24562.828,E2 -24562.828} C_VEL
LIN {X 0,Y 140.589,Z 392.864,A -85,B 0,C 180,E1 -24567.135,E2 -24567.135} C_VEL
LIN {X 0,Y 140.587,Z 394.597,A -85,B 0,C 180,E1 -24571.109,E2 -24571.109} C_VEL
LIN {X 0,Y 140.522,Z 395.206,A -85,B 0,C 180,E1 -24573.581,E2 -24573.581} C_VEL
LIN {X 0,Y 139.935,Z 395.59,A -85,B 0,C 180,E1 -24575.979,E2 -24575.979} C_VEL
LIN {X 0,Y 137.571,Z 395.516,A -85,B 0,C 180,E1 -24579.96,E2 -24579.96} C_VEL
LIN {X 0,Y 135.936,Z 395.05,A -85,B 0,C 180,E1 -24583.229,E2 -24583.229} C_VEL
LIN {X 0,Y 135.753,Z 394.437,A -85,B 0,C 180,E1 -24585.72,E2 -24585.72} C_VEL
LIN {X 0,Y 136.007,Z 394.126,A -85,B 0,C 180,E1 -24586.541,E2 -24586.541} C_VEL
LIN {X 0,Y 138.343,Z 392.259,A -85,B 0,C 180,E1 -24590.831,E2 -24590.831} C_VEL
LIN {X 0,Y 141.585,Z 389.394,A -85,B 0,C 180,E1 -24594.956,E2 -24594.956} C_VEL
LIN {X 0,Y 145.4,Z 385.552,A -85,B 0,C 180,E1 -24598.905,E2 -24598.905} C_VEL
LIN {X 0,Y 149.829,Z 380.639,A -85,B 0,C 180,E1 -24602.643,E2 -24602.643} C_VEL
LIN {X 0,Y 155.013,Z 374.52,A -85,B 0,C 180,E1 -24606.114,E2 -24606.114} C_VEL
LIN {X 0,Y 160.847,Z 366.969,A -85,B 0,C 180,E1 -24609.314,E2 -24609.314} C_VEL
LIN {X 0,Y 167.13,Z 357.57,A -85,B 0,C 180,E1 -24612.286,E2 -24612.286} C_VEL
LIN {X 0,Y 172.753,Z 347.938,A -85,B 0,C 180,E1 -24614.57,E2 -24614.57} C_VEL
LIN {X 0,Y 178.07,Z 337.297,A -85,B 0,C 180,E1 -24616.487,E2 -24616.487} C_VEL
LIN {X 0,Y 182.985,Z 325.31,A -85,B 0,C 180,E1 -24618.086,E2 -24618.086} C_VEL
LIN {X 0,Y 187.072,Z 312.794,A -85,B 0,C 180,E1 -24619.307,E2 -24619.307} C_VEL
LIN {X 0,Y 190.277,Z 299.705,A -85,B 0,C 180,E1 -24620.176,E2 -24620.176} C_VEL
LIN {X 0,Y 192.444,Z 285.462,A -85,B 0,C 180,E1 -24620.822,E2 -24620.822} C_VEL
LIN {X 0,Y 194.532,Z 264.155,A -85,B 0,C 180,E1 -24621.562,E2 -24621.562} C_VEL
LIN {X 0,Y 192.05,Z 257.119,A -85,B 0,C 180,E1 -24623.73,E2 -24623.73} C_VEL
LIN {X 0,Y 189.338,Z 250.496,A -85,B 0,C 180,E1 -24626.344,E2 -24626.344} C_VEL
LIN {X 0,Y 186.607,Z 244.41,A -85,B 0,C 180,E1 -24629.416,E2 -24629.416} C_VEL
LIN {X 0,Y 184.629,Z 240.233,A -85,B 0,C 180,E1 -24632.201,E2 -24632.201} C_VEL
LIN {X 0,Y 182.335,Z 235.563,A -85,B 0,C 180,E1 -24636.616,E2 -24636.616} C_VEL
LIN {X 0,Y 181.402,Z 234.48,A -85,B 0,C 180,E1 -24639.09,E2 -24639.09} C_VEL
LIN {X 0,Y 180.646,Z 233.587,A -85,B 0,C 180,E1 -24644.197,E2 -24644.197} C_VEL
LIN {X 0,Y 181.779,Z 234.422,A -85,B 0,C 180,E1 -24650.318,E2 -24650.318} C_VEL
LIN {X 0,Y 182.558,Z 235.114,A -85,B 0,C 180,E1 -24652.151,E2 -24652.151} C_VEL
LIN {X 0,Y 184.864,Z 238.986,A -85,B 0,C 180,E1 -24656.329,E2 -24656.329} C_VEL
LIN {X 0,Y 187.862,Z 244.317,A -85,B 0,C 180,E1 -24660.163,E2 -24660.163} C_VEL
LIN {X 0,Y 190.114,Z 248.445,A -85,B 0,C 180,E1 -24662.473,E2 -24662.473} C_VEL
LIN {X 0,Y 192.833,Z 253.861,A -85,B 0,C 180,E1 -24664.912,E2 -24664.912} C_VEL
LIN {X 0,Y 194.981,Z 259.276,A -85,B 0,C 180,E1 -24666.716,E2 -24666.716} C_VEL
LIN {X 0,Y 191.929,Z 287.584,A -85,B 0,C 180,E1 -24667.702,E2 -24667.702} C_VEL
LIN {X 0,Y 189.405,Z 300.978,A -85,B 0,C 180,E1 -24668.488,E2 -24668.488} C_VEL
LIN {X 0,Y 186.606,Z 311.488,A -85,B 0,C 180,E1 -24669.365,E2 -24669.365} C_VEL
LIN {X 0,Y 182.501,Z 323.704,A -85,B 0,C 180,E1 -24670.785,E2 -24670.785} C_VEL
LIN {X 0,Y 177.355,Z 335.708,A -85,B 0,C 180,E1 -24672.625,E2 -24672.625} C_VEL
LIN {X 0,Y 172.352,Z 345.411,A -85,B 0,C 180,E1 -24674.581,E2 -24674.581} C_VEL
LIN {X 0,Y 167.163,Z 354.087,A -85,B 0,C 180,E1 -24676.85,E2 -24676.85} C_VEL
LIN {X 0,Y 161.265,Z 362.607,A -85,B 0,C 180,E1 -24679.762,E2 -24679.762} C_VEL
LIN {X 0,Y 156.176,Z 369.156,A -85,B 0,C 180,E1 -24682.703,E2 -24682.703} C_VEL
LIN {X 0,Y 150.859,Z 375.281,A -85,B 0,C 180,E1 -24686.348,E2 -24686.348} C_VEL
LIN {X 0,Y 146.255,Z 380,A -85,B 0,C 180,E1 -24690.121,E2 -24690.121} C_VEL
LIN {X 0,Y 141.576,Z 384.26,A -85,B 0,C 180,E1 -24695.006,E2 -24695.006} C_VEL
LIN {X 0,Y 137.961,Z 386.987,A -85,B 0,C 180,E1 -24700.17,E2 -24700.17} C_VEL
LIN {X 0,Y 136.087,Z 388.063,A -85,B 0,C 180,E1 -24703.696,E2 -24703.696} C_VEL
LIN {X 0,Y 134.688,Z 388.527,A -85,B 0,C 180,E1 -24707.286,E2 -24707.286} C_VEL
LIN {X 0,Y 133.463,Z 388.264,A -85,B 0,C 180,E1 -24712.175,E2 -24712.175} C_VEL
LIN {X 0,Y 132.956,Z 386.575,A -85,B 0,C 180,E1 -24718.089,E2 -24718.089} C_VEL
LIN {X 0,Y 133.43,Z 383.615,A -85,B 0,C 180,E1 -24723.563,E2 -24723.563} C_VEL
LIN {X 0,Y 134.495,Z 379.581,A -85,B 0,C 180,E1 -24728.544,E2 -24728.544} C_VEL
LIN {X 0,Y 135.968,Z 374.143,A -85,B 0,C 180,E1 -24733.483,E2 -24733.483} C_VEL
LIN {X 0,Y 138.281,Z 367.182,A -85,B 0,C 180,E1 -24738.27,E2 -24738.27} C_VEL
LIN {X 0,Y 141.019,Z 359.384,A -85,B 0,C 180,E1 -24742.362,E2 -24742.362} C_VEL
LIN {X 0,Y 143.817,Z 351.102,A -85,B 0,C 180,E1 -24745.796,E2 -24745.796} C_VEL
LIN {X 0,Y 147.157,Z 340.808,A -85,B 0,C 180,E1 -24749.141,E2 -24749.141} C_VEL
LIN {X 0,Y 150.087,Z 330.775,A -85,B 0,C 180,E1 -24751.677,E2 -24751.677} C_VEL
LIN {X 0,Y 152.995,Z 319.106,A -85,B 0,C 180,E1 -24753.951,E2 -24753.951} C_VEL
LIN {X 0,Y 155.581,Z 306.53,A -85,B 0,C 180,E1 -24755.784,E2 -24755.784} C_VEL
LIN {X 0,Y 157.556,Z 293.938,A -85,B 0,C 180,E1 -24757.078,E2 -24757.078} C_VEL
LIN {X 0,Y 159.034,Z 280.137,A -85,B 0,C 180,E1 -24757.97,E2 -24757.97} C_VEL
LIN {X 0,Y 162.024,Z 235.95,A -85,B 0,C 180,E1 -24759.894,E2 -24759.894} C_VEL
LIN {X 0,Y 158.774,Z 226.335,A -85,B 0,C 180,E1 -24761.249,E2 -24761.249} C_VEL
LIN {X 0,Y 149.826,Z 208.912,A -85,B 0,C 180,E1 -24764.781,E2 -24764.781} C_VEL
LIN {X 0,Y 142.973,Z 197.914,A -85,B 0,C 180,E1 -24767.696,E2 -24767.696} C_VEL
LIN {X 0,Y 138.938,Z 191.411,A -85,B 0,C 180,E1 -24769.603,E2 -24769.603} C_VEL
LIN {X 0,Y 136.747,Z 188.514,A -85,B 0,C 180,E1 -24770.659,E2 -24770.659} C_VEL
LIN {X 0,Y 136.199,Z 186.517,A -85,B 0,C 180,E1 -24771.052,E2 -24771.052} C_VEL
LIN {X 0,Y 136.063,Z 186.537,A -85,B 0,C 180,E1 -24778.586,E2 -24778.586} C_VEL
LIN {X 0,Y 136.041,Z 186.505,A -85,B 0,C 180,E1 -24784.63,E2 -24784.63} C_VEL
LIN {X 0,Y 136.028,Z 186.542,A -85,B 0,C 180,E1 -24789.195,E2 -24789.195} C_VEL
LIN {X 0,Y 135.978,Z 186.511,A -85,B 0,C 180,E1 -24793.648,E2 -24793.648} C_VEL
LIN {X 0,Y 135.982,Z 186.496,A -85,B 0,C 180,E1 -24797.787,E2 -24797.787} C_VEL
LIN {X 0,Y 136.022,Z 186.533,A -85,B 0,C 180,E1 -24801.682,E2 -24801.682} C_VEL
LIN {X 0,Y 136.052,Z 186.533,A -85,B 0,C 180,E1 -24805.742,E2 -24805.742} C_VEL
LIN {X 0,Y 136.14,Z 186.527,A -85,B 0,C 180,E1 -24812.315,E2 -24812.315} C_VEL
LIN {X 0,Y 136.187,Z 186.513,A -85,B 0,C 180,E1 -24818.824,E2 -24818.824} C_VEL
LIN {X 0,Y 136.225,Z 186.498,A -85,B 0,C 180,E1 -24825.051,E2 -24825.051} C_VEL
LIN {X 0,Y 136.427,Z 186.486,A -85,B 0,C 180,E1 -24828.178,E2 -24828.178} C_VEL
LIN {X 0,Y 136.548,Z 186.473,A -85,B 0,C 180,E1 -24831.117,E2 -24831.117} C_VEL
LIN {X 0,Y 137.114,Z 186.402,A -85,B 0,C 180,E1 -24840,E2 -24840} C_VEL
LIN {X 0,Y 136.537,Z 186.432,A -85,B 0,C 180,E1 -24848.883,E2 -24848.883} C_VEL
LIN {X 0,Y 136.414,Z 186.485,A -85,B 0,C 180,E1 -24851.893,E2 -24851.893} C_VEL
LIN {X 0,Y 136.165,Z 186.494,A -85,B 0,C 180,E1 -24858.04,E2 -24858.04} C_VEL
LIN {X 0,Y 136.148,Z 186.488,A -85,B 0,C 180,E1 -24861.693,E2 -24861.693} C_VEL
LIN {X 0,Y 136.093,Z 186.524,A -85,B 0,C 180,E1 -24868.609,E2 -24868.609} C_VEL
LIN {X 0,Y 136.041,Z 186.536,A -85,B 0,C 180,E1 -24874.63,E2 -24874.63} C_VEL
LIN {X 0,Y 136.044,Z 186.542,A -85,B 0,C 180,E1 -24876.448,E2 -24876.448} C_VEL
LIN {X 0,Y 137.115,Z 189.548,A -85,B 0,C 180,E1 -24877.147,E2 -24877.147} C_VEL
LIN {X 0,Y 138.887,Z 191.754,A -85,B 0,C 180,E1 -24877.992,E2 -24877.992} C_VEL
LIN {X 0,Y 141.154,Z 195.247,A -85,B 0,C 180,E1 -24879.077,E2 -24879.077} C_VEL
LIN {X 0,Y 146.512,Z 204.238,A -85,B 0,C 180,E1 -24881.496,E2 -24881.496} C_VEL
LIN {X 0,Y 153.264,Z 219.211,A -85,B 0,C 180,E1 -24884.45,E2 -24884.45} C_VEL
LIN {X 0,Y 158.626,Z 233.592,A -85,B 0,C 180,E1 -24886.742,E2 -24886.742} C_VEL
LIN {X 0,Y 161.035,Z 241.361,A -85,B 0,C 180,E1 -24887.779,E2 -24887.779} C_VEL
LIN {X 0,Y 161.431,Z 247.976,A -85,B 0,C 180,E1 -24888.258,E2 -24888.258} C_VEL
LIN {X 0,Y 158.332,Z 292.916,A -85,B 0,C 180,E1 -24890.285,E2 -24890.285} C_VEL
LIN {X 0,Y 156.516,Z 306.666,A -85,B 0,C 180,E1 -24891.359,E2 -24891.359} C_VEL
LIN {X 0,Y 154.139,Z 319.279,A -85,B 0,C 180,E1 -24892.833,E2 -24892.833} C_VEL
LIN {X 0,Y 151.141,Z 331.739,A -85,B 0,C 180,E1 -24894.87,E2 -24894.87} C_VEL
LIN {X 0,Y 147.926,Z 342.913,A -85,B 0,C 180,E1 -24897.287,E2 -24897.287} C_VEL
LIN {X 0,Y 144.838,Z 353.028,A -85,B 0,C 180,E1 -24900.174,E2 -24900.174} C_VEL
LIN {X 0,Y 141.666,Z 362.152,A -85,B 0,C 180,E1 -24903.481,E2 -24903.481} C_VEL
LIN {X 0,Y 139.708,Z 368.348,A -85,B 0,C 180,E1 -24906.269,E2 -24906.269} C_VEL
LIN {X 0,Y 137.119,Z 375.981,A -85,B 0,C 180,E1 -24910.539,E2 -24910.539} C_VEL
LIN {X 0,Y 135.238,Z 382.096,A -85,B 0,C 180,E1 -24914.939,E2 -24914.939} C_VEL
LIN {X 0,Y 134.118,Z 386.914,A -85,B 0,C 180,E1 -24919.432,E2 -24919.432} C_VEL
LIN {X 0,Y 133.557,Z 390.562,A -85,B 0,C 180,E1 -24923.959,E2 -24923.959} C_VEL
LIN {X 0,Y 133.513,Z 392.429,A -85,B 0,C 180,E1 -24926.983,E2 -24926.983} C_VEL
LIN {X 0,Y 133.542,Z 394.051,A -85,B 0,C 180,E1 -24930.678,E2 -24930.678} C_VEL
LIN {X 0,Y 133.546,Z 395.316,A -85,B 0,C 180,E1 -24936.042,E2 -24936.042} C_VEL
LIN {X 0,Y 133.852,Z 395.493,A -85,B 0,C 180,E1 -24939.063,E2 -24939.063} C_VEL
LIN {X 0,Y 135.415,Z 394.634,A -85,B 0,C 180,E1 -24945.04,E2 -24945.04} C_VEL
LIN {X 0,Y 136.007,Z 394.126,A -85,B 0,C 180,E1 -24946.541,E2 -24946.541} C_VEL
LIN {X 0,Y 136.529,Z 393.258,A -85,B 0,C 180,E1 -24948.993,E2 -24948.993} C_VEL
LIN {X 0,Y 136.227,Z 391.348,A -85,B 0,C 180,E1 -24953.091,E2 -24953.091} C_VEL
LIN {X 0,Y 136.614,Z 388.801,A -85,B 0,C 180,E1 -24957.111,E2 -24957.111} C_VEL
LIN {X 0,Y 138.162,Z 386.85,A -85,B 0,C 180,E1 -24959.343,E2 -24959.343} C_VEL
LIN {X 0,Y 142.307,Z 382.816,A -85,B 0,C 180,E1 -24962.905,E2 -24962.905} C_VEL
LIN {X 0,Y 147.491,Z 377.284,A -85,B 0,C 180,E1 -24966.558,E2 -24966.558} C_VEL
LIN {X 0,Y 153.351,Z 370.43,A -85,B 0,C 180,E1 -24969.913,E2 -24969.913} C_VEL
LIN {X 0,Y 159.796,Z 361.911,A -85,B 0,C 180,E1 -24972.978,E2 -24972.978} C_VEL
LIN {X 0,Y 165.451,Z 353.261,A -85,B 0,C 180,E1 -24975.358,E2 -24975.358} C_VEL
LIN {X 0,Y 171.48,Z 342.728,A -85,B 0,C 180,E1 -24977.538,E2 -24977.538} C_VEL
LIN {X 0,Y 176.488,Z 332.323,A -85,B 0,C 180,E1 -24979.167,E2 -24979.167} C_VEL
LIN {X 0,Y 181.015,Z 320.839,A -85,B 0,C 180,E1 -24980.504,E2 -24980.504} C_VEL
LIN {X 0,Y 184.548,Z 309.673,A -85,B 0,C 180,E1 -24981.446,E2 -24981.446} C_VEL
LIN {X 0,Y 187.656,Z 296.189,A -85,B 0,C 180,E1 -24982.268,E2 -24982.268} C_VEL
LIN {X 0,Y 189.61,Z 282.058,A -85,B 0,C 180,E1 -24982.819,E2 -24982.819} C_VEL
LIN {X 0,Y 191.057,Z 267.114,A -85,B 0,C 180,E1 -24983.373,E2 -24983.373} C_VEL
LIN {X 0,Y 188.683,Z 260.314,A -85,B 0,C 180,E1 -24985.708,E2 -24985.708} C_VEL
LIN {X 0,Y 186.416,Z 254.474,A -85,B 0,C 180,E1 -24988.242,E2 -24988.242} C_VEL
LIN {X 0,Y 184.595,Z 250.281,A -85,B 0,C 180,E1 -24990.576,E2 -24990.576} C_VEL
LIN {X 0,Y 182.95,Z 246.565,A -85,B 0,C 180,E1 -24993.143,E2 -24993.143} C_VEL
LIN {X 0,Y 181.095,Z 242.344,A -85,B 0,C 180,E1 -24997.165,E2 -24997.165} C_VEL
LIN {X 0,Y 180.091,Z 241.211,A -85,B 0,C 180,E1 -25000.315,E2 -25000.315} C_VEL
LIN {X 0,Y 179.653,Z 240.627,A -85,B 0,C 180,E1 -25004.107,E2 -25004.107} C_VEL
LIN {X 0,Y 180.754,Z 241.451,A -85,B 0,C 180,E1 -25010.263,E2 -25010.263} C_VEL
LIN {X 0,Y 181.396,Z 242.157,A -85,B 0,C 180,E1 -25011.858,E2 -25011.858} C_VEL
LIN {X 0,Y 183.398,Z 245.743,A -85,B 0,C 180,E1 -25015.746,E2 -25015.746} C_VEL
LIN {X 0,Y 186.011,Z 250.624,A -85,B 0,C 180,E1 -25019.359,E2 -25019.359} C_VEL
LIN {X 0,Y 188.58,Z 255.638,A -85,B 0,C 180,E1 -25022.136,E2 -25022.136} C_VEL
LIN {X 0,Y 190.65,Z 260.376,A -85,B 0,C 180,E1 -25024.158,E2 -25024.158} C_VEL
LIN {X 0,Y 191.49,Z 262.789,A -85,B 0,C 180,E1 -25024.943,E2 -25024.943} C_VEL
LIN {X 0,Y 188.586,Z 288.34,A -85,B 0,C 180,E1 -25025.833,E2 -25025.833} C_VEL
LIN {X 0,Y 186.13,Z 300.826,A -85,B 0,C 180,E1 -25026.549,E2 -25026.549} C_VEL
LIN {X 0,Y 182.976,Z 312.323,A -85,B 0,C 180,E1 -25027.499,E2 -25027.499} C_VEL
LIN {X 0,Y 178.647,Z 324.475,A -85,B 0,C 180,E1 -25028.912,E2 -25028.912} C_VEL
LIN {X 0,Y 173.437,Z 336.046,A -85,B 0,C 180,E1 -25030.684,E2 -25030.684} C_VEL
LIN {X 0,Y 168.038,Z 345.992,A -85,B 0,C 180,E1 -25032.69,E2 -25032.69} C_VEL
LIN {X 0,Y 161.868,Z 355.627,A -85,B 0,C 180,E1 -25035.277,E2 -25035.277} C_VEL
LIN {X 0,Y 155.259,Z 364.537,A -85,B 0,C 180,E1 -25038.474,E2 -25038.474} C_VEL
LIN {X 0,Y 148.885,Z 371.998,A -85,B 0,C 180,E1 -25042.187,E2 -25042.187} C_VEL
LIN {X 0,Y 143.13,Z 377.871,A -85,B 0,C 180,E1 -25046.227,E2 -25046.227} C_VEL
LIN {X 0,Y 138.096,Z 382.378,A -85,B 0,C 180,E1 -25050.592,E2 -25050.592} C_VEL
LIN {X 0,Y 133.954,Z 385.616,A -85,B 0,C 180,E1 -25055.249,E2 -25055.249} C_VEL
LIN {X 0,Y 130.244,Z 387.914,A -85,B 0,C 180,E1 -25060.935,E2 -25060.935} C_VEL
LIN {X 0,Y 128.147,Z 388.71,A -85,B 0,C 180,E1 -25065.477,E2 -25065.477} C_VEL
LIN {X 0,Y 126.562,Z 388.514,A -85,B 0,C 180,E1 -25071.026,E2 -25071.026} C_VEL
LIN {X 0,Y 125.854,Z 387.02,A -85,B 0,C 180,E1 -25076.892,E2 -25076.892} C_VEL
LIN {X 0,Y 126.213,Z 384.047,A -85,B 0,C 180,E1 -25082.992,E2 -25082.992} C_VEL
LIN {X 0,Y 127.035,Z 380.99,A -85,B 0,C 180,E1 -25087.215,E2 -25087.215} C_VEL
LIN {X 0,Y 128.455,Z 375.936,A -85,B 0,C 180,E1 -25092.487,E2 -25092.487} C_VEL
LIN {X 0,Y 130.628,Z 369.358,A -85,B 0,C 180,E1 -25097.572,E2 -25097.572} C_VEL
LIN {X 0,Y 133.562,Z 361.325,A -85,B 0,C 180,E1 -25102.296,E2 -25102.296} C_VEL
LIN {X 0,Y 136.742,Z 352.431,A -85,B 0,C 180,E1 -25106.316,E2 -25106.316} C_VEL
LIN {X 0,Y 139.988,Z 342.93,A -85,B 0,C 180,E1 -25109.64,E2 -25109.64} C_VEL
LIN {X 0,Y 143.205,Z 332.609,A -85,B 0,C 180,E1 -25112.461,E2 -25112.461} C_VEL
LIN {X 0,Y 146.213,Z 321.463,A -85,B 0,C 180,E1 -25114.825,E2 -25114.825} C_VEL
LIN {X 0,Y 148.886,Z 309.297,A -85,B 0,C 180,E1 -25116.757,E2 -25116.757} C_VEL
LIN {X 0,Y 151.222,Z 295.771,A -85,B 0,C 180,E1 -25118.284,E2 -25118.284} C_VEL
LIN {X 0,Y 152.839,Z 282.551,A -85,B 0,C 180,E1 -25119.219,E2 -25119.219} C_VEL
LIN {X 0,Y 155.99,Z 237.45,A -85,B 0,C 180,E1 -25121.266,E2 -25121.266} C_VEL
LIN {X 0,Y 153.485,Z 229.962,A -85,B 0,C 180,E1 -25122.391,E2 -25122.391} C_VEL
LIN {X 0,Y 145.019,Z 213.222,A -85,B 0,C 180,E1 -25125.938,E2 -25125.938} C_VEL
LIN {X 0,Y 136.948,Z 200.011,A -85,B 0,C 180,E1 -25129.682,E2 -25129.682} C_VEL
LIN {X 0,Y 133.833,Z 195.46,A -85,B 0,C 180,E1 -25131.233,E2 -25131.233} C_VEL
LIN {X 0,Y 131.624,Z 192.042,A -85,B 0,C 180,E1 -25132.42,E2 -25132.42} C_VEL
LIN {X 0,Y 129.691,Z 189.708,A -85,B 0,C 180,E1 -25133.447,E2 -25133.447} C_VEL
LIN {X 0,Y 128.979,Z 187.393,A -85,B 0,C 180,E1 -25133.983,E2 -25133.983} C_VEL
LIN {X 0,Y 129,Z 187.413,A -85,B 0,C 180,E1 -25139.362,E2 -25139.362} C_VEL
LIN {X 0,Y 128.957,Z 187.389,A -85,B 0,C 180,E1 -25145.166,E2 -25145.166} C_VEL
LIN {X 0,Y 128.924,Z 187.421,A -85,B 0,C 180,E1 -25150.856,E2 -25150.856} C_VEL
LIN {X 0,Y 128.912,Z 187.374,A -85,B 0,C 180,E1 -25155.132,E2 -25155.132} C_VEL
LIN {X 0,Y 128.934,Z 187.394,A -85,B 0,C 180,E1 -25159.74,E2 -25159.74} C_VEL
LIN {X 0,Y 128.957,Z 187.42,A -85,B 0,C 180,E1 -25164.834,E2 -25164.834} C_VEL
LIN {X 0,Y 129.018,Z 187.41,A -85,B 0,C 180,E1 -25170.642,E2 -25170.642} C_VEL
LIN {X 0,Y 129.011,Z 187.409,A -85,B 0,C 180,E1 -25174.163,E2 -25174.163} C_VEL
LIN {X 0,Y 129.07,Z 187.393,A -85,B 0,C 180,E1 -25177.77,E2 -25177.77} C_VEL
LIN {X 0,Y 129.147,Z 187.382,A -85,B 0,C 180,E1 -25184.211,E2 -25184.211} C_VEL
LIN {X 0,Y 129.344,Z 187.368,A -85,B 0,C 180,E1 -25187.972,E2 -25187.972} C_VEL
LIN {X 0,Y 129.471,Z 187.356,A -85,B 0,C 180,E1 -25190.628,E2 -25190.628} C_VEL
LIN {X 0,Y 130.069,Z 187.279,A -85,B 0,C 180,E1 -25200,E2 -25200} C_VEL
LIN {X 0,Y 129.462,Z 187.316,A -85,B 0,C 180,E1 -25209.373,E2 -25209.373} C_VEL
LIN {X 0,Y 129.298,Z 187.375,A -85,B 0,C 180,E1 -25212.557,E2 -25212.557} C_VEL
LIN {X 0,Y 129.081,Z 187.365,A -85,B 0,C 180,E1 -25219.067,E2 -25219.067} C_VEL
LIN {X 0,Y 129.044,Z 187.377,A -85,B 0,C 180,E1 -25222.41,E2 -25222.41} C_VEL
LIN {X 0,Y 129.009,Z 187.416,A -85,B 0,C 180,E1 -25225.837,E2 -25225.837} C_VEL
LIN {X 0,Y 129.018,Z 187.406,A -85,B 0,C 180,E1 -25229.358,E2 -25229.358} C_VEL
LIN {X 0,Y 128.998,Z 187.412,A -85,B 0,C 180,E1 -25233.602,E2 -25233.602} C_VEL
LIN {X 0,Y 130.05,Z 190.33,A -85,B 0,C 180,E1 -25234.355,E2 -25234.355} C_VEL
LIN {X 0,Y 132.099,Z 192.879,A -85,B 0,C 180,E1 -25235.435,E2 -25235.435} C_VEL
LIN {X 0,Y 134.217,Z 196.156,A -85,B 0,C 180,E1 -25236.558,E2 -25236.558} C_VEL
LIN {X 0,Y 141.026,Z 207.027,A -85,B 0,C 180,E1 -25239.904,E2 -25239.904} C_VEL
LIN {X 0,Y 147.615,Z 221.718,A -85,B 0,C 180,E1 -25243.02,E2 -25243.02} C_VEL
LIN {X 0,Y 153.07,Z 236.461,A -85,B 0,C 180,E1 -25245.503,E2 -25245.503} C_VEL
LIN {X 0,Y 155.2,Z 243.534,A -85,B 0,C 180,E1 -25246.499,E2 -25246.499} C_VEL
LIN {X 0,Y 155.418,Z 249.076,A -85,B 0,C 180,E1 -25246.897,E2 -25246.897} C_VEL
LIN {X 0,Y 152.295,Z 292.41,A -85,B 0,C 180,E1 -25248.897,E2 -25248.897} C_VEL
LIN {X 0,Y 150.52,Z 305.695,A -85,B 0,C 180,E1 -25249.949,E2 -25249.949} C_VEL
LIN {X 0,Y 148.066,Z 318.567,A -85,B 0,C 180,E1 -25251.465,E2 -25251.465} C_VEL
LIN {X 0,Y 144.936,Z 331.135,A -85,B 0,C 180,E1 -25253.558,E2 -25253.558} C_VEL
LIN {X 0,Y 141.557,Z 342.376,A -85,B 0,C 180,E1 -25256.045,E2 -25256.045} C_VEL
LIN {X 0,Y 138.651,Z 351.547,A -85,B 0,C 180,E1 -25258.697,E2 -25258.697} C_VEL
LIN {X 0,Y 136.104,Z 359.021,A -85,B 0,C 180,E1 -25261.382,E2 -25261.382} C_VEL
LIN {X 0,Y 133.22,Z 367.253,A -85,B 0,C 180,E1 -25265.036,E2 -25265.036} C_VEL
LIN {X 0,Y 130.427,Z 375.077,A -85,B 0,C 180,E1 -25269.497,E2 -25269.497} C_VEL
LIN {X 0,Y 128.354,Z 381.324,A -85,B 0,C 180,E1 -25274.111,E2 -25274.111} C_VEL
LIN {X 0,Y 127.127,Z 386.267,A -85,B 0,C 180,E1 -25278.843,E2 -25278.843} C_VEL
LIN {X 0,Y 126.507,Z 390.031,A -85,B 0,C 180,E1 -25283.621,E2 -25283.621} C_VEL
LIN {X 0,Y 126.439,Z 391.956,A -85,B 0,C 180,E1 -25286.814,E2 -25286.814} C_VEL
LIN {X 0,Y 126.504,Z 393.434,A -85,B 0,C 180,E1 -25290,E2 -25290} C_VEL
LIN {X 0,Y 126.375,Z 394.431,A -85,B 0,C 180,E1 -25293.188,E2 -25293.188} C_VEL
LIN {X 0,Y 126.844,Z 395.269,A -85,B 0,C 180,E1 -25299.568,E2 -25299.568} C_VEL
LIN {X 0,Y 127.506,Z 395.124,A -85,B 0,C 180,E1 -25302.737,E2 -25302.737} C_VEL
LIN {X 0,Y 129.897,Z 393.632,A -85,B 0,C 180,E1 -25308.943,E2 -25308.943} C_VEL
LIN {X 0,Y 133.951,Z 390.597,A -85,B 0,C 180,E1 -25314.818,E2 -25314.818} C_VEL
LIN {X 0,Y 138.162,Z 386.85,A -85,B 0,C 180,E1 -25319.343,E2 -25319.343} C_VEL
LIN {X 0,Y 139.075,Z 385.477,A -85,B 0,C 180,E1 -25320.847,E2 -25320.847} C_VEL
LIN {X 0,Y 139.283,Z 380.935,A -85,B 0,C 180,E1 -25326.093,E2 -25326.093} C_VEL
LIN {X 0,Y 140.558,Z 379.15,A -85,B 0,C 180,E1 -25327.451,E2 -25327.451} C_VEL
LIN {X 0,Y 146.964,Z 372.37,A -85,B 0,C 180,E1 -25331.113,E2 -25331.113} C_VEL
LIN {X 0,Y 153.565,Z 364.419,A -85,B 0,C 180,E1 -25334.261,E2 -25334.261} C_VEL
LIN {X 0,Y 160.602,Z 354.608,A -85,B 0,C 180,E1 -25337.138,E2 -25337.138} C_VEL
LIN {X 0,Y 166.838,Z 344.379,A -85,B 0,C 180,E1 -25339.31,E2 -25339.31} C_VEL
LIN {X 0,Y 172.67,Z 332.978,A -85,B 0,C 180,E1 -25341.117,E2 -25341.117} C_VEL
LIN {X 0,Y 177.349,Z 321.793,A -85,B 0,C 180,E1 -25342.426,E2 -25342.426} C_VEL
LIN {X 0,Y 181.095,Z 310.558,A -85,B 0,C 180,E1 -25343.379,E2 -25343.379} C_VEL
LIN {X 0,Y 184.451,Z 296.773,A -85,B 0,C 180,E1 -25344.209,E2 -25344.209} C_VEL
LIN {X 0,Y 186.556,Z 282.699,A -85,B 0,C 180,E1 -25344.758,E2 -25344.758} C_VEL
LIN {X 0,Y 187.827,Z 270.395,A -85,B 0,C 180,E1 -25345.203,E2 -25345.203} C_VEL
LIN {X 0,Y 185.624,Z 263.703,A -85,B 0,C 180,E1 -25347.733,E2 -25347.733} C_VEL
LIN {X 0,Y 183.577,Z 258.326,A -85,B 0,C 180,E1 -25350.397,E2 -25350.397} C_VEL
LIN {X 0,Y 181.528,Z 253.257,A -85,B 0,C 180,E1 -25353.739,E2 -25353.739} C_VEL
LIN {X 0,Y 179.895,Z 249.178,A -85,B 0,C 180,E1 -25357.647,E2 -25357.647} C_VEL
LIN {X 0,Y 178.997,Z 248.115,A -85,B 0,C 180,E1 -25360.817,E2 -25360.817} C_VEL
LIN {X 0,Y 178.66,Z 247.668,A -85,B 0,C 180,E1 -25364.016,E2 -25364.016} C_VEL
LIN {X 0,Y 179.517,Z 248.323,A -85,B 0,C 180,E1 -25369.626,E2 -25369.626} C_VEL
LIN {X 0,Y 180.184,Z 249.017,A -85,B 0,C 180,E1 -25371.398,E2 -25371.398} C_VEL
LIN {X 0,Y 181.952,Z 252.455,A -85,B 0,C 180,E1 -25375.148,E2 -25375.148} C_VEL
LIN {X 0,Y 184.242,Z 257.027,A -85,B 0,C 180,E1 -25378.557,E2 -25378.557} C_VEL
LIN {X 0,Y 186.378,Z 261.449,A -85,B 0,C 180,E1 -25381.08,E2 -25381.08} C_VEL
LIN {X 0,Y 188.222,Z 265.965,A -85,B 0,C 180,E1 -25383.051,E2 -25383.051} C_VEL
LIN {X 0,Y 186.627,Z 281.183,A -85,B 0,C 180,E1 -25383.598,E2 -25383.598} C_VEL
LIN {X 0,Y 184.516,Z 294.261,A -85,B 0,C 180,E1 -25384.153,E2 -25384.153} C_VEL
LIN {X 0,Y 181.235,Z 307.571,A -85,B 0,C 180,E1 -25385.041,E2 -25385.041} C_VEL
LIN {X 0,Y 177.201,Z 319.737,A -85,B 0,C 180,E1 -25386.27,E2 -25386.27} C_VEL
LIN {X 0,Y 171.925,Z 332.09,A -85,B 0,C 180,E1 -25387.933,E2 -25387.933} C_VEL
LIN {X 0,Y 166.023,Z 343.15,A -85,B 0,C 180,E1 -25389.937,E2 -25389.937} C_VEL
LIN {X 0,Y 159.994,Z 352.621,A -85,B 0,C 180,E1 -25392.211,E2 -25392.211} C_VEL
LIN {X 0,Y 152.986,Z 362.047,A -85,B 0,C 180,E1 -25395.264,E2 -25395.264} C_VEL
LIN {X 0,Y 145.743,Z 370.332,A -85,B 0,C 180,E1 -25399.032,E2 -25399.032} C_VEL
LIN {X 0,Y 139.417,Z 376.687,A -85,B 0,C 180,E1 -25403.075,E2 -25403.075} C_VEL
LIN {X 0,Y 134.205,Z 381.213,A -85,B 0,C 180,E1 -25407.094,E2 -25407.094} C_VEL
LIN {X 0,Y 130.523,Z 384.001,A -85,B 0,C 180,E1 -25410.511,E2 -25410.511} C_VEL
LIN {X 0,Y 127.369,Z 386.173,A -85,B 0,C 180,E1 -25414.139,E2 -25414.139} C_VEL
LIN {X 0,Y 124.363,Z 387.868,A -85,B 0,C 180,E1 -25418.436,E2 -25418.436} C_VEL
LIN {X 0,Y 121.554,Z 388.9,A -85,B 0,C 180,E1 -25423.933,E2 -25423.933} C_VEL
LIN {X 0,Y 119.714,Z 388.759,A -85,B 0,C 180,E1 -25429.776,E2 -25429.776} C_VEL
LIN {X 0,Y 118.816,Z 387.338,A -85,B 0,C 180,E1 -25435.905,E2 -25435.905} C_VEL
LIN {X 0,Y 119.007,Z 384.44,A -85,B 0,C 180,E1 -25442.355,E2 -25442.355} C_VEL
LIN {X 0,Y 119.992,Z 380.894,A -85,B 0,C 180,E1 -25447.572,E2 -25447.572} C_VEL
LIN {X 0,Y 121.53,Z 375.67,A -85,B 0,C 180,E1 -25453.193,E2 -25453.193} C_VEL
LIN {X 0,Y 123.851,Z 368.977,A -85,B 0,C 180,E1 -25458.544,E2 -25458.544} C_VEL
LIN {X 0,Y 126.506,Z 362.052,A -85,B 0,C 180,E1 -25462.819,E2 -25462.819} C_VEL
LIN {X 0,Y 129.648,Z 353.666,A -85,B 0,C 180,E1 -25466.892,E2 -25466.892} C_VEL
LIN {X 0,Y 133.218,Z 343.805,A -85,B 0,C 180,E1 -25470.574,E2 -25470.574} C_VEL
LIN {X 0,Y 136.783,Z 332.946,A -85,B 0,C 180,E1 -25473.682,E2 -25473.682} C_VEL
LIN {X 0,Y 140.096,Z 321.1,A -85,B 0,C 180,E1 -25476.271,E2 -25476.271} C_VEL
LIN {X 0,Y 142.979,Z 308.439,A -85,B 0,C 180,E1 -25478.299,E2 -25478.299} C_VEL
LIN {X 0,Y 145.232,Z 295.82,A -85,B 0,C 180,E1 -25479.738,E2 -25479.738} C_VEL
LIN {X 0,Y 146.874,Z 282.806,A -85,B 0,C 180,E1 -25480.684,E2 -25480.684} C_VEL
LIN {X 0,Y 150.02,Z 238.807,A -85,B 0,C 180,E1 -25482.756,E2 -25482.756} C_VEL
LIN {X 0,Y 148.104,Z 233.302,A -85,B 0,C 180,E1 -25483.646,E2 -25483.646} C_VEL
LIN {X 0,Y 140.388,Z 217.743,A -85,B 0,C 180,E1 -25487.12,E2 -25487.12} C_VEL
LIN {X 0,Y 132.624,Z 204.819,A -85,B 0,C 180,E1 -25490.948,E2 -25490.948} C_VEL
LIN {X 0,Y 127.535,Z 197.222,A -85,B 0,C 180,E1 -25493.748,E2 -25493.748} C_VEL
LIN {X 0,Y 125.29,Z 193.922,A -85,B 0,C 180,E1 -25495.088,E2 -25495.088} C_VEL
LIN {X 0,Y 124.596,Z 192.983,A -85,B 0,C 180,E1 -25495.511,E2 -25495.511} C_VEL
LIN {X 0,Y 122.641,Z 190.663,A -85,B 0,C 180,E1 -25496.717,E2 -25496.717} C_VEL
LIN {X 0,Y 121.873,Z 188.301,A -85,B 0,C 180,E1 -25497.473,E2 -25497.473} C_VEL
LIN {X 0,Y 121.891,Z 188.275,A -85,B 0,C 180,E1 -25501.26,E2 -25501.26} C_VEL
LIN {X 0,Y 121.882,Z 188.278,A -85,B 0,C 180,E1 -25506.169,E2 -25506.169} C_VEL
LIN {X 0,Y 121.864,Z 188.295,A -85,B 0,C 180,E1 -25511.434,E2 -25511.434} C_VEL
LIN {X 0,Y 121.846,Z 188.259,A -85,B 0,C 180,E1 -25518.576,E2 -25518.576} C_VEL
LIN {X 0,Y 121.908,Z 188.298,A -85,B 0,C 180,E1 -25524.795,E2 -25524.795} C_VEL
LIN {X 0,Y 121.927,Z 188.287,A -85,B 0,C 180,E1 -25529.839,E2 -25529.839} C_VEL
LIN {X 0,Y 121.952,Z 188.276,A -85,B 0,C 180,E1 -25536.209,E2 -25536.209} C_VEL
LIN {X 0,Y 121.99,Z 188.287,A -85,B 0,C 180,E1 -25539.777,E2 -25539.777} C_VEL
LIN {X 0,Y 122.188,Z 188.249,A -85,B 0,C 180,E1 -25546.698,E2 -25546.698} C_VEL
LIN {X 0,Y 122.397,Z 188.239,A -85,B 0,C 180,E1 -25550.081,E2 -25550.081} C_VEL
LIN {X 0,Y 122.564,Z 188.212,A -85,B 0,C 180,E1 -25556.713,E2 -25556.713} C_VEL
LIN {X 0,Y 123.022,Z 188.157,A -85,B 0,C 180,E1 -25560,E2 -25560} C_VEL
LIN {X 0,Y 122.405,Z 188.173,A -85,B 0,C 180,E1 -25566.594,E2 -25566.594} C_VEL
LIN {X 0,Y 122.391,Z 188.202,A -85,B 0,C 180,E1 -25569.92,E2 -25569.92} C_VEL
LIN {X 0,Y 122.187,Z 188.264,A -85,B 0,C 180,E1 -25573.301,E2 -25573.301} C_VEL
LIN {X 0,Y 121.986,Z 188.244,A -85,B 0,C 180,E1 -25580.223,E2 -25580.223} C_VEL
LIN {X 0,Y 121.951,Z 188.276,A -85,B 0,C 180,E1 -25583.791,E2 -25583.791} C_VEL
LIN {X 0,Y 121.912,Z 188.295,A -85,B 0,C 180,E1 -25590.251,E2 -25590.251} C_VEL
LIN {X 0,Y 122.809,Z 191.002,A -85,B 0,C 180,E1 -25591,E2 -25591} C_VEL
LIN {X 0,Y 125.219,Z 193.754,A -85,B 0,C 180,E1 -25592.458,E2 -25592.458} C_VEL
LIN {X 0,Y 127.332,Z 197.082,A -85,B 0,C 180,E1 -25593.74,E2 -25593.74} C_VEL
LIN {X 0,Y 133.136,Z 206.004,A -85,B 0,C 180,E1 -25596.933,E2 -25596.933} C_VEL
LIN {X 0,Y 137.335,Z 213.287,A -85,B 0,C 180,E1 -25599.074,E2 -25599.074} C_VEL
LIN {X 0,Y 143.585,Z 228.139,A -85,B 0,C 180,E1 -25602.248,E2 -25602.248} C_VEL
LIN {X 0,Y 149.052,Z 243.798,A -85,B 0,C 180,E1 -25604.889,E2 -25604.889} C_VEL
LIN {X 0,Y 149.622,Z 248,A -85,B 0,C 180,E1 -25605.319,E2 -25605.319} C_VEL
LIN {X 0,Y 146.337,Z 292.261,A -85,B 0,C 180,E1 -25607.425,E2 -25607.425} C_VEL
LIN {X 0,Y 144.502,Z 305.462,A -85,B 0,C 180,E1 -25608.496,E2 -25608.496} C_VEL
LIN {X 0,Y 142.07,Z 317.799,A -85,B 0,C 180,E1 -25609.977,E2 -25609.977} C_VEL
LIN {X 0,Y 139.288,Z 328.941,A -85,B 0,C 180,E1 -25611.823,E2 -25611.823} C_VEL
LIN {X 0,Y 135.631,Z 340.495,A -85,B 0,C 180,E1 -25614.342,E2 -25614.342} C_VEL
LIN {X 0,Y 132.933,Z 348.871,A -85,B 0,C 180,E1 -25616.735,E2 -25616.735} C_VEL
LIN {X 0,Y 129.622,Z 358.397,A -85,B 0,C 180,E1 -25620.171,E2 -25620.171} C_VEL
LIN {X 0,Y 127.258,Z 364.732,A -85,B 0,C 180,E1 -25622.992,E2 -25622.992} C_VEL
LIN {X 0,Y 124.205,Z 372.882,A -85,B 0,C 180,E1 -25627.546,E2 -25627.546} C_VEL
LIN {X 0,Y 122.112,Z 378.523,A -85,B 0,C 180,E1 -25631.546,E2 -25631.546} C_VEL
LIN {X 0,Y 120.498,Z 384.028,A -85,B 0,C 180,E1 -25636.509,E2 -25636.509} C_VEL
LIN {X 0,Y 119.601,Z 388.296,A -85,B 0,C 180,E1 -25641.552,E2 -25641.552} C_VEL
LIN {X 0,Y 119.354,Z 391.454,A -85,B 0,C 180,E1 -25646.624,E2 -25646.624} C_VEL
LIN {X 0,Y 119.417,Z 393.001,A -85,B 0,C 180,E1 -25650,E2 -25650} C_VEL
LIN {X 0,Y 119.283,Z 394.095,A -85,B 0,C 180,E1 -25653.378,E2 -25653.378} C_VEL
LIN {X 0,Y 119.415,Z 394.76,A -85,B 0,C 180,E1 -25656.76,E2 -25656.76} C_VEL
LIN {X 0,Y 120.568,Z 394.954,A -85,B 0,C 180,E1 -25663.484,E2 -25663.484} C_VEL
LIN {X 0,Y 121.708,Z 394.494,A -85,B 0,C 180,E1 -25666.782,E2 -25666.782} C_VEL
LIN {X 0,Y 123.176,Z 393.631,A -85,B 0,C 180,E1 -25670.02,E2 -25670.02} C_VEL
LIN {X 0,Y 127.547,Z 390.728,A -85,B 0,C 180,E1 -25676.156,E2 -25676.156} C_VEL
LIN {X 0,Y 131.82,Z 387.303,A -85,B 0,C 180,E1 -25680.672,E2 -25680.672} C_VEL
LIN {X 0,Y 136.405,Z 383.218,A -85,B 0,C 180,E1 -25684.525,E2 -25684.525} C_VEL
LIN {X 0,Y 140.558,Z 379.15,A -85,B 0,C 180,E1 -25687.451,E2 -25687.451} C_VEL
LIN {X 0,Y 141.935,Z 377.299,A -85,B 0,C 180,E1 -25688.776,E2 -25688.776} C_VEL
LIN {X 0,Y 143.842,Z 371.393,A -85,B 0,C 180,E1 -25693.596,E2 -25693.596} C_VEL
LIN {X 0,Y 145.427,Z 369.145,A -85,B 0,C 180,E1 -25694.733,E2 -25694.733} C_VEL
LIN {X 0,Y 152.237,Z 360.874,A -85,B 0,C 180,E1 -25697.616,E2 -25697.616} C_VEL
LIN {X 0,Y 158.484,Z 352.128,A -85,B 0,C 180,E1 -25699.904,E2 -25699.904} C_VEL
LIN {X 0,Y 165.041,Z 341.446,A -85,B 0,C 180,E1 -25701.98,E2 -25701.98} C_VEL
LIN {X 0,Y 170.434,Z 330.83,A -85,B 0,C 180,E1 -25703.524,E2 -25703.524} C_VEL
LIN {X 0,Y 175.271,Z 319.128,A -85,B 0,C 180,E1 -25704.786,E2 -25704.786} C_VEL
LIN {X 0,Y 179.362,Z 306.603,A -85,B 0,C 180,E1 -25705.712,E2 -25705.712} C_VEL
LIN {X 0,Y 182.265,Z 293.838,A -85,B 0,C 180,E1 -25706.396,E2 -25706.396} C_VEL
LIN {X 0,Y 184.706,Z 275.232,A -85,B 0,C 180,E1 -25707.052,E2 -25707.052} C_VEL
LIN {X 0,Y 184.787,Z 273.542,A -85,B 0,C 180,E1 -25707.195,E2 -25707.195} C_VEL
LIN {X 0,Y 182.609,Z 266.725,A -85,B 0,C 180,E1 -25710.112,E2 -25710.112} C_VEL
LIN {X 0,Y 180.984,Z 262.272,A -85,B 0,C 180,E1 -25712.727,E2 -25712.727} C_VEL
LIN {X 0,Y 179.92,Z 259.467,A -85,B 0,C 180,E1 -25714.79,E2 -25714.79} C_VEL
LIN {X 0,Y 178.669,Z 255.968,A -85,B 0,C 180,E1 -25718.241,E2 -25718.241} C_VEL
LIN {X 0,Y 177.754,Z 254.855,A -85,B 0,C 180,E1 -25722.541,E2 -25722.541} C_VEL
LIN {X 0,Y 177.981,Z 254.933,A -85,B 0,C 180,E1 -25727.415,E2 -25727.415} C_VEL
LIN {X 0,Y 178.963,Z 255.794,A -85,B 0,C 180,E1 -25730.863,E2 -25730.863} C_VEL
LIN {X 0,Y 180.558,Z 259.266,A -85,B 0,C 180,E1 -25734.606,E2 -25734.606} C_VEL
LIN {X 0,Y 182.695,Z 263.75,A -85,B 0,C 180,E1 -25737.976,E2 -25737.976} C_VEL
LIN {X 0,Y 185.168,Z 269.524,A -85,B 0,C 180,E1 -25741.087,E2 -25741.087} C_VEL
LIN {X 0,Y 185.209,Z 270.47,A -85,B 0,C 180,E1 -25741.238,E2 -25741.238} C_VEL
LIN {X 0,Y 182.658,Z 289.89,A -85,B 0,C 180,E1 -25741.879,E2 -25741.879} C_VEL
LIN {X 0,Y 179.862,Z 302.602,A -85,B 0,C 180,E1 -25742.591,E2 -25742.591} C_VEL
LIN {X 0,Y 176.44,Z 313.801,A -85,B 0,C 180,E1 -25743.509,E2 -25743.509} C_VEL
LIN {X 0,Y 171.492,Z 326.33,A -85,B 0,C 180,E1 -25744.946,E2 -25744.946} C_VEL
LIN {X 0,Y 166.24,Z 336.939,A -85,B 0,C 180,E1 -25746.546,E2 -25746.546} C_VEL
LIN {X 0,Y 159.946,Z 347.411,A -85,B 0,C 180,E1 -25748.638,E2 -25748.638} C_VEL
LIN {X 0,Y 153.603,Z 356.364,A -85,B 0,C 180,E1 -25751.017,E2 -25751.017} C_VEL
LIN {X 0,Y 147.05,Z 364.326,A -85,B 0,C 180,E1 -25753.826,E2 -25753.826} C_VEL
LIN {X 0,Y 139.795,Z 371.977,A -85,B 0,C 180,E1 -25757.556,E2 -25757.556} C_VEL
LIN {X 0,Y 133.235,Z 377.913,A -85,B 0,C 180,E1 -25761.669,E2 -25761.669} C_VEL
LIN {X 0,Y 127.302,Z 382.517,A -85,B 0,C 180,E1 -25766.21,E2 -25766.21} C_VEL
LIN {X 0,Y 122.269,Z 385.855,A -85,B 0,C 180,E1 -25771.153,E2 -25771.153} C_VEL
LIN {X 0,Y 118.214,Z 388.02,A -85,B 0,C 180,E1 -25776.478,E2 -25776.478} C_VEL
LIN {X 0,Y 114.819,Z 389.126,A -85,B 0,C 180,E1 -25782.733,E2 -25782.733} C_VEL
LIN {X 0,Y 112.911,Z 389.005,A -85,B 0,C 180,E1 -25788.325,E2 -25788.325} C_VEL
LIN {X 0,Y 111.792,Z 387.645,A -85,B 0,C 180,E1 -25794.813,E2 -25794.813} C_VEL
LIN {X 0,Y 111.811,Z 384.828,A -85,B 0,C 180,E1 -25801.642,E2 -25801.642} C_VEL
LIN {X 0,Y 112.974,Z 380.711,A -85,B 0,C 180,E1 -25808.083,E2 -25808.083} C_VEL
LIN {X 0,Y 114.61,Z 375.387,A -85,B 0,C 180,E1 -25813.981,E2 -25813.981} C_VEL
LIN {X 0,Y 117.105,Z 368.585,A -85,B 0,C 180,E1 -25819.628,E2 -25819.628} C_VEL
LIN {X 0,Y 120.08,Z 361.285,A -85,B 0,C 180,E1 -25824.256,E2 -25824.256} C_VEL
LIN {X 0,Y 123.328,Z 352.962,A -85,B 0,C 180,E1 -25828.367,E2 -25828.367} C_VEL
LIN {X 0,Y 127.121,Z 342.876,A -85,B 0,C 180,E1 -25832.185,E2 -25832.185} C_VEL
LIN {X 0,Y 130.856,Z 331.807,A -85,B 0,C 180,E1 -25835.393,E2 -25835.393} C_VEL
LIN {X 0,Y 133.989,Z 320.968,A -85,B 0,C 180,E1 -25837.775,E2 -25837.775} C_VEL
LIN {X 0,Y 136.885,Z 308.733,A -85,B 0,C 180,E1 -25839.792,E2 -25839.792} C_VEL
LIN {X 0,Y 139.241,Z 296.069,A -85,B 0,C 180,E1 -25841.279,E2 -25841.279} C_VEL
LIN {X 0,Y 141,Z 282.736,A -85,B 0,C 180,E1 -25842.261,E2 -25842.261} C_VEL
LIN {X 0,Y 144.181,Z 240.602,A -85,B 0,C 180,E1 -25844.286,E2 -25844.286} C_VEL
LIN {X 0,Y 142.781,Z 236.715,A -85,B 0,C 180,E1 -25844.98,E2 -25844.98} C_VEL
LIN {X 0,Y 135.805,Z 222.246,A -85,B 0,C 180,E1 -25848.374,E2 -25848.374} C_VEL
LIN {X 0,Y 128.443,Z 209.768,A -85,B 0,C 180,E1 -25852.254,E2 -25852.254} C_VEL
LIN {X 0,Y 123.565,Z 202.353,A -85,B 0,C 180,E1 -25855.141,E2 -25855.141} C_VEL
LIN {X 0,Y 120.859,Z 198.456,A -85,B 0,C 180,E1 -25856.87,E2 -25856.87} C_VEL
LIN {X 0,Y 118.602,Z 195.326,A -85,B 0,C 180,E1 -25858.397,E2 -25858.397} C_VEL
LIN {X 0,Y 117.848,Z 194.148,A -85,B 0,C 180,E1 -25858.946,E2 -25858.946} C_VEL
LIN {X 0,Y 115.746,Z 191.805,A -85,B 0,C 180,E1 -25860.429,E2 -25860.429} C_VEL
LIN {X 0,Y 114.853,Z 189.148,A -85,B 0,C 180,E1 -25861.397,E2 -25861.397} C_VEL
LIN {X 0,Y 114.777,Z 189.181,A -85,B 0,C 180,E1 -25867.758,E2 -25867.758} C_VEL
LIN {X 0,Y 114.779,Z 189.156,A -85,B 0,C 180,E1 -25872.712,E2 -25872.712} C_VEL
LIN {X 0,Y 114.769,Z 189.131,A -85,B 0,C 180,E1 -25877.655,E2 -25877.655} C_VEL
LIN {X 0,Y 114.785,Z 189.184,A -85,B 0,C 180,E1 -25882.747,E2 -25882.747} C_VEL
LIN {X 0,Y 114.855,Z 189.161,A -85,B 0,C 180,E1 -25888.944,E2 -25888.944} C_VEL
LIN {X 0,Y 114.915,Z 189.152,A -85,B 0,C 180,E1 -25896.546,E2 -25896.546} C_VEL
LIN {X 0,Y 114.966,Z 189.161,A -85,B 0,C 180,E1 -25902.202,E2 -25902.202} C_VEL
LIN {X 0,Y 115.31,Z 189.121,A -85,B 0,C 180,E1 -25909.464,E2 -25909.464} C_VEL
LIN {X 0,Y 115.49,Z 189.092,A -85,B 0,C 180,E1 -25916.511,E2 -25916.511} C_VEL
LIN {X 0,Y 115.974,Z 189.034,A -85,B 0,C 180,E1 -25920,E2 -25920} C_VEL
LIN {X 0,Y 115.347,Z 189.051,A -85,B 0,C 180,E1 -25926.999,E2 -25926.999} C_VEL
LIN {X 0,Y 115.204,Z 189.129,A -85,B 0,C 180,E1 -25932.556,E2 -25932.556} C_VEL
LIN {X 0,Y 114.964,Z 189.131,A -85,B 0,C 180,E1 -25937.798,E2 -25937.798} C_VEL
LIN {X 0,Y 114.914,Z 189.145,A -85,B 0,C 180,E1 -25943.452,E2 -25943.452} C_VEL
LIN {X 0,Y 114.868,Z 189.257,A -85,B 0,C 180,E1 -25946.332,E2 -25946.332} C_VEL
LIN {X 0,Y 115.81,Z 191.911,A -85,B 0,C 180,E1 -25947.196,E2 -25947.196} C_VEL
LIN {X 0,Y 117.91,Z 194.163,A -85,B 0,C 180,E1 -25948.672,E2 -25948.672} C_VEL
LIN {X 0,Y 120.704,Z 198.334,A -85,B 0,C 180,E1 -25950.614,E2 -25950.614} C_VEL
LIN {X 0,Y 122.006,Z 200.162,A -85,B 0,C 180,E1 -25951.469,E2 -25951.469} C_VEL
LIN {X 0,Y 125.172,Z 204.984,A -85,B 0,C 180,E1 -25953.457,E2 -25953.457} C_VEL
LIN {X 0,Y 131.382,Z 215.054,A -85,B 0,C 180,E1 -25956.984,E2 -25956.984} C_VEL
LIN {X 0,Y 134.901,Z 222.685,A -85,B 0,C 180,E1 -25958.916,E2 -25958.916} C_VEL
LIN {X 0,Y 139.581,Z 234.796,A -85,B 0,C 180,E1 -25961.452,E2 -25961.452} C_VEL
LIN {X 0,Y 143.692,Z 247.319,A -85,B 0,C 180,E1 -25963.616,E2 -25963.616} C_VEL
LIN {X 0,Y 143.634,Z 251.348,A -85,B 0,C 180,E1 -25963.877,E2 -25963.877} C_VEL
LIN {X 0,Y 140.402,Z 292.375,A -85,B 0,C 180,E1 -25965.885,E2 -25965.885} C_VEL
LIN {X 0,Y 138.327,Z 306.352,A -85,B 0,C 180,E1 -25967.067,E2 -25967.067} C_VEL
LIN {X 0,Y 135.663,Z 318.864,A -85,B 0,C 180,E1 -25968.661,E2 -25968.661} C_VEL
LIN {X 0,Y 132.295,Z 331.283,A -85,B 0,C 180,E1 -25970.887,E2 -25970.887} C_VEL
LIN {X 0,Y 128.656,Z 342.421,A -85,B 0,C 180,E1 -25973.554,E2 -25973.554} C_VEL
LIN {X 0,Y 125.038,Z 352.709,A -85,B 0,C 180,E1 -25976.865,E2 -25976.865} C_VEL
LIN {X 0,Y 121.959,Z 360.567,A -85,B 0,C 180,E1 -25980.059,E2 -25980.059} C_VEL
LIN {X 0,Y 119.186,Z 367.802,A -85,B 0,C 180,E1 -25983.752,E2 -25983.752} C_VEL
LIN {X 0,Y 116.209,Z 375.424,A -85,B 0,C 180,E1 -25988.724,E2 -25988.724} C_VEL
LIN {X 0,Y 114.074,Z 381.53,A -85,B 0,C 180,E1 -25993.904,E2 -25993.904} C_VEL
LIN {X 0,Y 112.841,Z 386.338,A -85,B 0,C 180,E1 -25999.231,E2 -25999.231} C_VEL
LIN {X 0,Y 112.285,Z 389.974,A -85,B 0,C 180,E1 -26004.613,E2 -26004.613} C_VEL
LIN {X 0,Y 112.332,Z 392.554,A -85,B 0,C 180,E1 -26010,E2 -26010} C_VEL
LIN {X 0,Y 112.201,Z 393.722,A -85,B 0,C 180,E1 -26013.591,E2 -26013.591} C_VEL
LIN {X 0,Y 112.347,Z 394.479,A -85,B 0,C 180,E1 -26017.187,E2 -26017.187} C_VEL
LIN {X 0,Y 113.66,Z 394.786,A -85,B 0,C 180,E1 -26024.32,E2 -26024.32} C_VEL
LIN {X 0,Y 116.504,Z 393.619,A -85,B 0,C 180,E1 -26031.22,E2 -26031.22} C_VEL
LIN {X 0,Y 118.643,Z 392.448,A -85,B 0,C 180,E1 -26034.498,E2 -26034.498} C_VEL
LIN {X 0,Y 121.203,Z 390.866,A -85,B 0,C 180,E1 -26037.638,E2 -26037.638} C_VEL
LIN {X 0,Y 125.551,Z 387.744,A -85,B 0,C 180,E1 -26042.126,E2 -26042.126} C_VEL
LIN {X 0,Y 130.624,Z 383.635,A -85,B 0,C 180,E1 -26046.288,E2 -26046.288} C_VEL
LIN {X 0,Y 136.413,Z 378.428,A -85,B 0,C 180,E1 -26050.091,E2 -26050.091} C_VEL
LIN {X 0,Y 142.844,Z 371.944,A -85,B 0,C 180,E1 -26053.536,E2 -26053.536} C_VEL
LIN {X 0,Y 145.427,Z 369.145,A -85,B 0,C 180,E1 -26054.733,E2 -26054.733} C_VEL
LIN {X 0,Y 147.042,Z 366.84,A -85,B 0,C 180,E1 -26055.843,E2 -26055.843} C_VEL
LIN {X 0,Y 149.813,Z 359.639,A -85,B 0,C 180,E1 -26060.146,E2 -26060.146} C_VEL
LIN {X 0,Y 151.521,Z 356.993,A -85,B 0,C 180,E1 -26061.065,E2 -26061.065} C_VEL
LIN {X 0,Y 158.775,Z 346.602,A -85,B 0,C 180,E1 -26063.349,E2 -26063.349} C_VEL
LIN {X 0,Y 165.002,Z 335.891,A -85,B 0,C 180,E1 -26065.078,E2 -26065.078} C_VEL
LIN {X 0,Y 170.67,Z 323.856,A -85,B 0,C 180,E1 -26066.499,E2 -26066.499} C_VEL
LIN {X 0,Y 175.047,Z 312.211,A -85,B 0,C 180,E1 -26067.473,E2 -26067.473} C_VEL
LIN {X 0,Y 178.698,Z 299.02,A -85,B 0,C 180,E1 -26068.264,E2 -26068.264} C_VEL
LIN {X 0,Y 181.214,Z 284.729,A -85,B 0,C 180,E1 -26068.832,E2 -26068.832} C_VEL
LIN {X 0,Y 182.037,Z 277.323,A -85,B 0,C 180,E1 -26069.108,E2 -26069.108} C_VEL
LIN {X 0,Y 180.631,Z 272.4,A -85,B 0,C 180,E1 -26071.366,E2 -26071.366} C_VEL
LIN {X 0,Y 179.27,Z 268.266,A -85,B 0,C 180,E1 -26073.845,E2 -26073.845} C_VEL
LIN {X 0,Y 178.439,Z 265.801,A -85,B 0,C 180,E1 -26075.773,E2 -26075.773} C_VEL
LIN {X 0,Y 177.46,Z 262.722,A -85,B 0,C 180,E1 -26078.861,E2 -26078.861} C_VEL
LIN {X 0,Y 176.669,Z 261.747,A -85,B 0,C 180,E1 -26083.831,E2 -26083.831} C_VEL
LIN {X 0,Y 177.368,Z 262.292,A -85,B 0,C 180,E1 -26089.159,E2 -26089.159} C_VEL
LIN {X 0,Y 177.89,Z 263.012,A -85,B 0,C 180,E1 -26090.777,E2 -26090.777} C_VEL
LIN {X 0,Y 179.158,Z 265.911,A -85,B 0,C 180,E1 -26093.941,E2 -26093.941} C_VEL
LIN {X 0,Y 181.387,Z 270.95,A -85,B 0,C 180,E1 -26097.709,E2 -26097.709} C_VEL
LIN {X 0,Y 182.399,Z 273.65,A -85,B 0,C 180,E1 -26099.181,E2 -26099.181} C_VEL
LIN {X 0,Y 180.12,Z 290.469,A -85,B 0,C 180,E1 -26099.802,E2 -26099.802} C_VEL
LIN {X 0,Y 177.199,Z 303.163,A -85,B 0,C 180,E1 -26100.489,E2 -26100.489} C_VEL
LIN {X 0,Y 173.658,Z 314.307,A -85,B 0,C 180,E1 -26101.381,E2 -26101.381} C_VEL
LIN {X 0,Y 168.86,Z 326.097,A -85,B 0,C 180,E1 -26102.69,E2 -26102.69} C_VEL
LIN {X 0,Y 162.994,Z 337.54,A -85,B 0,C 180,E1 -26104.353,E2 -26104.353} C_VEL
LIN {X 0,Y 156.447,Z 347.937,A -85,B 0,C 180,E1 -26106.398,E2 -26106.398} C_VEL
LIN {X 0,Y 149.384,Z 357.351,A -85,B 0,C 180,E1 -26108.89,E2 -26108.89} C_VEL
LIN {X 0,Y 141.895,Z 365.852,A -85,B 0,C 180,E1 -26111.98,E2 -26111.98} C_VEL
LIN {X 0,Y 133.943,Z 373.526,A -85,B 0,C 180,E1 -26115.961,E2 -26115.961} C_VEL
LIN {X 0,Y 127.205,Z 379.093,A -85,B 0,C 180,E1 -26120.075,E2 -26120.075} C_VEL
LIN {X 0,Y 120.279,Z 383.891,A -85,B 0,C 180,E1 -26125.369,E2 -26125.369} C_VEL
LIN {X 0,Y 114.777,Z 387.007,A -85,B 0,C 180,E1 -26130.991,E2 -26130.991} C_VEL
LIN {X 0,Y 111.681,Z 388.404,A -85,B 0,C 180,E1 -26135.106,E2 -26135.106} C_VEL
LIN {X 0,Y 108.649,Z 389.273,A -85,B 0,C 180,E1 -26140.305,E2 -26140.305} C_VEL
LIN {X 0,Y 106.17,Z 389.235,A -85,B 0,C 180,E1 -26146.732,E2 -26146.732} C_VEL
LIN {X 0,Y 104.812,Z 387.939,A -85,B 0,C 180,E1 -26153.576,E2 -26153.576} C_VEL
LIN {X 0,Y 104.646,Z 385.197,A -85,B 0,C 180,E1 -26160.819,E2 -26160.819} C_VEL
LIN {X 0,Y 105.459,Z 382.015,A -85,B 0,C 180,E1 -26166.431,E2 -26166.431} C_VEL
LIN {X 0,Y 107.015,Z 377.056,A -85,B 0,C 180,E1 -26172.811,E2 -26172.811} C_VEL
LIN {X 0,Y 109.423,Z 370.671,A -85,B 0,C 180,E1 -26178.89,E2 -26178.89} C_VEL
LIN {X 0,Y 112.299,Z 363.686,A -85,B 0,C 180,E1 -26183.92,E2 -26183.92} C_VEL
LIN {X 0,Y 115.574,Z 355.931,A -85,B 0,C 180,E1 -26188.258,E2 -26188.258} C_VEL
LIN {X 0,Y 119.596,Z 345.937,A -85,B 0,C 180,E1 -26192.56,E2 -26192.56} C_VEL
LIN {X 0,Y 123.646,Z 334.872,A -85,B 0,C 180,E1 -26196.118,E2 -26196.118} C_VEL
LIN {X 0,Y 127.057,Z 324.1,A -85,B 0,C 180,E1 -26198.749,E2 -26198.749} C_VEL
LIN {X 0,Y 130.124,Z 312.512,A -85,B 0,C 180,E1 -26200.896,E2 -26200.896} C_VEL
LIN {X 0,Y 132.733,Z 299.99,A -85,B 0,C 180,E1 -26202.567,E2 -26202.567} C_VEL
LIN {X 0,Y 134.82,Z 286.145,A -85,B 0,C 180,E1 -26203.776,E2 -26203.776} C_VEL
LIN {X 0,Y 138.511,Z 242.603,A -85,B 0,C 180,E1 -26205.911,E2 -26205.911} C_VEL
LIN {X 0,Y 136.998,Z 239.004,A -85,B 0,C 180,E1 -26206.685,E2 -26206.685} C_VEL
LIN {X 0,Y 131.2,Z 226.603,A -85,B 0,C 180,E1 -26209.725,E2 -26209.725} C_VEL
LIN {X 0,Y 124.265,Z 214.596,A -85,B 0,C 180,E1 -26213.686,E2 -26213.686} C_VEL
LIN {X 0,Y 119.79,Z 207.636,A -85,B 0,C 180,E1 -26216.517,E2 -26216.517} C_VEL
LIN {X 0,Y 117.026,Z 203.665,A -85,B 0,C 180,E1 -26218.412,E2 -26218.412} C_VEL
LIN {X 0,Y 114.206,Z 199.63,A -85,B 0,C 180,E1 -26220.511,E2 -26220.511} C_VEL
LIN {X 0,Y 111.935,Z 196.486,A -85,B 0,C 180,E1 -26222.323,E2 -26222.323} C_VEL
LIN {X 0,Y 111.218,Z 195.26,A -85,B 0,C 180,E1 -26222.954,E2 -26222.954} C_VEL
LIN {X 0,Y 108.915,Z 193.176,A -85,B 0,C 180,E1 -26224.858,E2 -26224.858} C_VEL
LIN {X 0,Y 107.853,Z 190.792,A -85,B 0,C 180,E1 -26225.974,E2 -26225.974} C_VEL
LIN {X 0,Y 107.721,Z 190.039,A -85,B 0,C 180,E1 -26226.301,E2 -26226.301} C_VEL
LIN {X 0,Y 107.676,Z 190.067,A -85,B 0,C 180,E1 -26230.746,E2 -26230.746} C_VEL
LIN {X 0,Y 107.658,Z 190.012,A -85,B 0,C 180,E1 -26235.897,E2 -26235.897} C_VEL
LIN {X 0,Y 107.681,Z 190.058,A -85,B 0,C 180,E1 -26241.555,E2 -26241.555} C_VEL
LIN {X 0,Y 107.792,Z 190.039,A -85,B 0,C 180,E1 -26248.56,E2 -26248.56} C_VEL
LIN {X 0,Y 107.831,Z 190.035,A -85,B 0,C 180,E1 -26255.85,E2 -26255.85} C_VEL
LIN {X 0,Y 107.864,Z 190.049,A -85,B 0,C 180,E1 -26260.987,E2 -26260.987} C_VEL
LIN {X 0,Y 108.227,Z 190.001,A -85,B 0,C 180,E1 -26268.766,E2 -26268.766} C_VEL
LIN {X 0,Y 108.293,Z 189.982,A -85,B 0,C 180,E1 -26272.542,E2 -26272.542} C_VEL
LIN {X 0,Y 108.9,Z 189.915,A -85,B 0,C 180,E1 -26280,E2 -26280} C_VEL
LIN {X 0,Y 108.287,Z 189.929,A -85,B 0,C 180,E1 -26287.458,E2 -26287.458} C_VEL
LIN {X 0,Y 108.138,Z 190.011,A -85,B 0,C 180,E1 -26292.872,E2 -26292.872} C_VEL
LIN {X 0,Y 107.886,Z 190,A -85,B 0,C 180,E1 -26301.495,E2 -26301.495} C_VEL
LIN {X 0,Y 108.862,Z 192.859,A -85,B 0,C 180,E1 -26302.664,E2 -26302.664} C_VEL
LIN {X 0,Y 111.024,Z 195.118,A -85,B 0,C 180,E1 -26304.494,E2 -26304.494} C_VEL
LIN {X 0,Y 111.748,Z 196.096,A -85,B 0,C 180,E1 -26305.1,E2 -26305.1} C_VEL
LIN {X 0,Y 113.875,Z 199.294,A -85,B 0,C 180,E1 -26306.827,E2 -26306.827} C_VEL
LIN {X 0,Y 114.994,Z 200.585,A -85,B 0,C 180,E1 -26307.652,E2 -26307.652} C_VEL
LIN {X 0,Y 117.573,Z 204.301,A -85,B 0,C 180,E1 -26309.54,E2 -26309.54} C_VEL
LIN {X 0,Y 122.891,Z 212.677,A -85,B 0,C 180,E1 -26313.086,E2 -26313.086} C_VEL
LIN {X 0,Y 127.882,Z 221.346,A -85,B 0,C 180,E1 -26316.091,E2 -26316.091} C_VEL
LIN {X 0,Y 133.523,Z 235.405,A -85,B 0,C 180,E1 -26319.413,E2 -26319.413} C_VEL
LIN {X 0,Y 137.964,Z 248.866,A -85,B 0,C 180,E1 -26321.958,E2 -26321.958} C_VEL
LIN {X 0,Y 137.703,Z 254.842,A -85,B 0,C 180,E1 -26322.313,E2 -26322.313} C_VEL
LIN {X 0,Y 134.677,Z 291.622,A -85,B 0,C 180,E1 -26324.149,E2 -26324.149} C_VEL
LIN {X 0,Y 132.665,Z 305.044,A -85,B 0,C 180,E1 -26325.284,E2 -26325.284} C_VEL
LIN {X 0,Y 129.878,Z 317.908,A -85,B 0,C 180,E1 -26326.908,E2 -26326.908} C_VEL
LIN {X 0,Y 126.364,Z 330.493,A -85,B 0,C 180,E1 -26329.194,E2 -26329.194} C_VEL
LIN {X 0,Y 122.519,Z 341.728,A -85,B 0,C 180,E1 -26331.928,E2 -26331.928} C_VEL
LIN {X 0,Y 118.789,Z 351.941,A -85,B 0,C 180,E1 -26335.288,E2 -26335.288} C_VEL
LIN {X 0,Y 115.552,Z 359.903,A -85,B 0,C 180,E1 -26338.624,E2 -26338.624} C_VEL
LIN {X 0,Y 112.207,Z 368.031,A -85,B 0,C 180,E1 -26342.993,E2 -26342.993} C_VEL
LIN {X 0,Y 109.12,Z 375.58,A -85,B 0,C 180,E1 -26348.264,E2 -26348.264} C_VEL
LIN {X 0,Y 106.687,Z 382.512,A -85,B 0,C 180,E1 -26354.722,E2 -26354.722} C_VEL
LIN {X 0,Y 105.541,Z 387.038,A -85,B 0,C 180,E1 -26360.417,E2 -26360.417} C_VEL
LIN {X 0,Y 105.184,Z 390.436,A -85,B 0,C 180,E1 -26366.169,E2 -26366.169} C_VEL
LIN {X 0,Y 105.262,Z 392.098,A -85,B 0,C 180,E1 -26370,E2 -26370} C_VEL
LIN {X 0,Y 105.113,Z 393.318,A -85,B 0,C 180,E1 -26373.834,E2 -26373.834} C_VEL
LIN {X 0,Y 105.289,Z 394.149,A -85,B 0,C 180,E1 -26377.672,E2 -26377.672} C_VEL
LIN {X 0,Y 105.831,Z 394.589,A -85,B 0,C 180,E1 -26381.492,E2 -26381.492} C_VEL
